FUNCTION_BLOCK "LProcModeSelector"   // FB1708, FBD
TITLE = LModeSelector
{ S7_Optimized_Access := 'FALSE' }
AUTHOR : VCC
FAMILY : Control
NAME : ModeSel
VERSION : 1.0
// ================================================================================
// This module handles that only one mode is selected in the modezon, it also 
// handle interlocking between the HMIs. Each modezone can have 5 HMI.
// ================================================================================
// stored: AutoNumber false, IsIECCheckEnabled false, SetENOAutomatically False, UDAEnableTagReadback false
   VAR_INPUT
      I_StartPB { ExternalAccessible := 'False'; ExternalVisible := 'False'; ExternalWritable := 'False'} : Bool;   // Summary of Start buttons
      I_AlarmResetPB { ExternalAccessible := 'False'; ExternalVisible := 'False'; ExternalWritable := 'False'} : Bool;   // Summary of Alarm reset buttons
      I_SafetyNotOk { ExternalAccessible := 'False'; ExternalVisible := 'False'; ExternalWritable := 'False'} : Bool;   // Safety is not ok
      I_FailSafeResetAck { ExternalAccessible := 'False'; ExternalVisible := 'False'; ExternalWritable := 'False'} : Bool;   // F_Ack_Op FB in safety program is requesting value 9 on FailSafeReset output
      I_FailSafeAckID { ExternalAccessible := 'False'; ExternalVisible := 'False'; ExternalWritable := 'False'} : Int;   // F_Ack ID
      I_HMI1ForceMan { ExternalAccessible := 'False'; ExternalVisible := 'False'; ExternalWritable := 'False'} : Bool;   // Forced manual selected on HMI1
      I_HMI1SetPB { ExternalAccessible := 'False'; ExternalVisible := 'False'; ExternalWritable := 'False'} : Bool;   // Set PB activated on HMI1
      I_HMI1ResetPB { ExternalAccessible := 'False'; ExternalVisible := 'False'; ExternalWritable := 'False'} : Bool;   // Reset PB activated on HMI1
      I_HMI1StartPB { ExternalAccessible := 'False'; ExternalVisible := 'False'; ExternalWritable := 'False'} : Bool;   // Start PB activated on HMI1
      I_HMI1AlarmResetPB { ExternalAccessible := 'False'; ExternalVisible := 'False'; ExternalWritable := 'False'} : Bool;   // AlarmReset PB activated on HMI1
      I_HMI2ForceMan { ExternalAccessible := 'False'; ExternalVisible := 'False'; ExternalWritable := 'False'} : Bool;   // Forced manual selected on HMI2
      I_HMI2SetPB { ExternalAccessible := 'False'; ExternalVisible := 'False'; ExternalWritable := 'False'} : Bool;   // Set PB activated on HMI2
      I_HMI2ResetPB { ExternalAccessible := 'False'; ExternalVisible := 'False'; ExternalWritable := 'False'} : Bool;   // Reset PB activated on HMI2
      I_HMI2StartPB { ExternalAccessible := 'False'; ExternalVisible := 'False'; ExternalWritable := 'False'} : Bool;   // Start PB activated on HMI2
      I_HMI2AlarmResetPB { ExternalAccessible := 'False'; ExternalVisible := 'False'; ExternalWritable := 'False'} : Bool;   // AlarmReset PB activated on HMI2
      I_HMI3ForceMan { ExternalAccessible := 'False'; ExternalVisible := 'False'; ExternalWritable := 'False'} : Bool;   // Forced manual selected on HMI3
      I_HMI3SetPB { ExternalAccessible := 'False'; ExternalVisible := 'False'; ExternalWritable := 'False'} : Bool;   // Set PB activated on HMI3
      I_HMI3ResetPB { ExternalAccessible := 'False'; ExternalVisible := 'False'; ExternalWritable := 'False'} : Bool;   // Reset PB activated on HMI3
      I_HMI3StartPB { ExternalAccessible := 'False'; ExternalVisible := 'False'; ExternalWritable := 'False'} : Bool;   // Start PB activated on HMI
      I_HMI3AlarmResetPB { ExternalAccessible := 'False'; ExternalVisible := 'False'; ExternalWritable := 'False'} : Bool;   // AlarmReset PB activated on HMI3
      I_HMI4ForceMan { ExternalAccessible := 'False'; ExternalVisible := 'False'; ExternalWritable := 'False'} : Bool;   // Forced manual selected on HMI4
      I_HMI4SetPB { ExternalAccessible := 'False'; ExternalVisible := 'False'; ExternalWritable := 'False'} : Bool;   // Set PB activated on HMI4
      I_HMI4ResetPB { ExternalAccessible := 'False'; ExternalVisible := 'False'; ExternalWritable := 'False'} : Bool;   // Reset PB activated on HMI4
      I_HMI4StartPB { ExternalAccessible := 'False'; ExternalVisible := 'False'; ExternalWritable := 'False'} : Bool;   // Start PB activated on HMI4
      I_HMI4AlarmResetPB { ExternalAccessible := 'False'; ExternalVisible := 'False'; ExternalWritable := 'False'} : Bool;   // AlarmReset PB activated on HMI4
      I_HMI5ForceMan { ExternalAccessible := 'False'; ExternalVisible := 'False'; ExternalWritable := 'False'} : Bool;   // Forced manual selected on HMI5
      I_HMI5SetPB { ExternalAccessible := 'False'; ExternalVisible := 'False'; ExternalWritable := 'False'} : Bool;   // Set PB activated on HMI5
      I_HMI5ResetPB { ExternalAccessible := 'False'; ExternalVisible := 'False'; ExternalWritable := 'False'} : Bool;   // Reset PB activated on HMI5
      I_HMI5StartPB { ExternalAccessible := 'False'; ExternalVisible := 'False'; ExternalWritable := 'False'} : Bool;   // Start PB activated on HMI5
      I_HMI5AlarmResetPB { ExternalAccessible := 'False'; ExternalVisible := 'False'; ExternalWritable := 'False'} : Bool;   // AlarmReset PB activated on HMI5
   END_VAR
   VAR_OUTPUT
      O_PBSetPBResetAllAutoSel { ExternalAccessible := 'False'; ExternalVisible := 'False'; ExternalWritable := 'False'} : Struct   // Set PB activated - Reset PB activated - All HMI Auto selected
         HMI1SetPB { ExternalAccessible := 'False'; ExternalVisible := 'False'; ExternalWritable := 'False'} : Bool;   // Set PB activated on HMI1
         HMI1ResetPB { ExternalAccessible := 'False'; ExternalVisible := 'False'; ExternalWritable := 'False'} : Bool;   // Reset PB activated on HMI1
         HMI1AllHMIAutoSel { ExternalAccessible := 'False'; ExternalVisible := 'False'; ExternalWritable := 'False'} : Bool;   // All HMI Auto selected on HMI1
         HMI2SetPB { ExternalAccessible := 'False'; ExternalVisible := 'False'; ExternalWritable := 'False'} : Bool;   // Set PB activated on HMI2
         HMI2ResetPB { ExternalAccessible := 'False'; ExternalVisible := 'False'; ExternalWritable := 'False'} : Bool;   // Reset PB activated on HMI2
         HMI2AllHMIAutoSel { ExternalAccessible := 'False'; ExternalVisible := 'False'; ExternalWritable := 'False'} : Bool;   // All HMI Auto selected on HMI2
         HMI3SetPB { ExternalAccessible := 'False'; ExternalVisible := 'False'; ExternalWritable := 'False'} : Bool;   // Set PB activated on HMI3
         HMI3ResetPB { ExternalAccessible := 'False'; ExternalVisible := 'False'; ExternalWritable := 'False'} : Bool;   // Reset PB activated on HMI3
         HMI3AllHMIAutoSel { ExternalAccessible := 'False'; ExternalVisible := 'False'; ExternalWritable := 'False'} : Bool;   // All HMI Auto selected on HMI3
         HMI4SetPB { ExternalAccessible := 'False'; ExternalVisible := 'False'; ExternalWritable := 'False'} : Bool;   // Set PB activated on HMI4
         HMI4ResetPB { ExternalAccessible := 'False'; ExternalVisible := 'False'; ExternalWritable := 'False'} : Bool;   // Reset PB activated on HMI4
         HMI4AllHMIAutoSel { ExternalAccessible := 'False'; ExternalVisible := 'False'; ExternalWritable := 'False'} : Bool;   // All HMI Auto selected on HMI4
         HMI5SetPB { ExternalAccessible := 'False'; ExternalVisible := 'False'; ExternalWritable := 'False'} : Bool;   // Set PB activated on HMI5
         HMI5ResetPB { ExternalAccessible := 'False'; ExternalVisible := 'False'; ExternalWritable := 'False'} : Bool;   // Reset PB activated on HMI5
         HMI5AllHMIAutoSel { ExternalAccessible := 'False'; ExternalVisible := 'False'; ExternalWritable := 'False'} : Bool;   // All HMI Auto selected on HMI5
         StartPBSel { ExternalAccessible := 'False'; ExternalVisible := 'False'; ExternalWritable := 'False'} : Bool;   // Start is activated
         AlarmResetPBSel { ExternalAccessible := 'False'; ExternalVisible := 'False'; ExternalWritable := 'False'} : Bool;   // Alarm reset is activated
      END_STRUCT;
   END_VAR
   VAR_IN_OUT
      IO_FailsafeReset { ExternalAccessible := 'False'; ExternalVisible := 'False'; ExternalWritable := 'False'} : Int;   // Number to Failsafe to reset safety
   END_VAR
   VAR DB_SPECIFIC
      H_HMIHomeRunModeCmd : Word;   // Homerun Mode commands from HMI
      H_Anim : Word;   // Animation for HMI
      H_ActiveHMI : Int;   // Active HMI
      H_NameActiveHMI : String[25];   // Name of the Active HMI
      H_LockManTime : Int;   // Lock manual time
      H_HMI1ModeCmd : Word;   // Mode commands from HMI1
      H_HMI2ModeCmd : Word;   // Mode commands from HMI2
      H_HMI3ModeCmd : Word;   // Mode commands from HMI3
      H_HMI4ModeCmd : Word;   // Mode commands from HMI4
      H_HMI5ModeCmd : Word;   // Mode commands from HMI5. For operator panels, no S7_m_c
      HMI1AutoSel { ExternalAccessible := 'False'; ExternalVisible := 'False'; ExternalWritable := 'False'} : Bool;   // Auto selected on HMI1
      HMI1StepSel { ExternalAccessible := 'False'; ExternalVisible := 'False'; ExternalWritable := 'False'} : Bool;   // Step selected on HMI1
      HMI1HomeRunSel { ExternalAccessible := 'False'; ExternalVisible := 'False'; ExternalWritable := 'False'} : Bool;   // Homerun selected on HMI1
      HMI1ManualSel { ExternalAccessible := 'False'; ExternalVisible := 'False'; ExternalWritable := 'False'} : Bool;   // Manual selected on HMI1
      HMI1LockManual { ExternalAccessible := 'False'; ExternalVisible := 'False'; ExternalWritable := 'False'} : Bool;   // Lock manual for HMI1
      HMI1AllHMIAutoSel { ExternalAccessible := 'False'; ExternalVisible := 'False'; ExternalWritable := 'False'} : Bool;   // All HMI Auto selected on HMI1
      HMI1Start { ExternalAccessible := 'False'; ExternalVisible := 'False'; ExternalWritable := 'False'} : Bool;   // Start on HMI1
      HMI1AlarmReset { ExternalAccessible := 'False'; ExternalVisible := 'False'; ExternalWritable := 'False'} : Bool;   // AlarmReset on HMI1
      HMI1ResetTM { ExternalAccessible := 'False'; ExternalVisible := 'False'; ExternalWritable := 'False'} : Bool;   // Reset transport memory from HMI1
      HMI1ResetSeq { ExternalAccessible := 'False'; ExternalVisible := 'False'; ExternalWritable := 'False'} : Bool;   // Reset sequence from HMI1
      HMI1CycleFinished { ExternalAccessible := 'False'; ExternalVisible := 'False'; ExternalWritable := 'False'} : Bool;   // Cycle Finished from HMI1
      HMI1AlarmResetAck { ExternalAccessible := 'False'; ExternalVisible := 'False'; ExternalWritable := 'False'} : Bool;   // Alarm Reset acknowledge from HMI1
      HMI2AutoSel { ExternalAccessible := 'False'; ExternalVisible := 'False'; ExternalWritable := 'False'} : Bool;   // Auto selected on HMI2
      HMI2StepSel { ExternalAccessible := 'False'; ExternalVisible := 'False'; ExternalWritable := 'False'} : Bool;   // Step selected on HMI2
      HMI2HomeRunSel { ExternalAccessible := 'False'; ExternalVisible := 'False'; ExternalWritable := 'False'} : Bool;   // Homerun selected on HMI2
      HMI2ManualSel { ExternalAccessible := 'False'; ExternalVisible := 'False'; ExternalWritable := 'False'} : Bool;   // Manual selected on HMI2
      HMI2LockManual { ExternalAccessible := 'False'; ExternalVisible := 'False'; ExternalWritable := 'False'} : Bool;   // Lock manual for HMI2
      HMI2AllHMIAutoSel { ExternalAccessible := 'False'; ExternalVisible := 'False'; ExternalWritable := 'False'} : Bool;   // All HMI Auto selected on HMI2
      HMI2Start { ExternalAccessible := 'False'; ExternalVisible := 'False'; ExternalWritable := 'False'} : Bool;   // Start on HMI2
      HMI2AlarmReset { ExternalAccessible := 'False'; ExternalVisible := 'False'; ExternalWritable := 'False'} : Bool;   // AlarmReset on HMI2
      HMI2ResetTM { ExternalAccessible := 'False'; ExternalVisible := 'False'; ExternalWritable := 'False'} : Bool;   // Reset transport memory from HMI2
      HMI2ResetSeq { ExternalAccessible := 'False'; ExternalVisible := 'False'; ExternalWritable := 'False'} : Bool;   // Reset sequence from HMI2
      HMI2CycleFinished { ExternalAccessible := 'False'; ExternalVisible := 'False'; ExternalWritable := 'False'} : Bool;   // Cycle Finished from HMI2
      HMI2AlarmResetAck { ExternalAccessible := 'False'; ExternalVisible := 'False'; ExternalWritable := 'False'} : Bool;   // Alarm Reset acknowledge from HMI2
      HMI3AutoSel { ExternalAccessible := 'False'; ExternalVisible := 'False'; ExternalWritable := 'False'} : Bool;   // Auto selected on HMI3
      HMI3StepSel { ExternalAccessible := 'False'; ExternalVisible := 'False'; ExternalWritable := 'False'} : Bool;   // Step selected on HMI3
      HMI3HomeRunSel { ExternalAccessible := 'False'; ExternalVisible := 'False'; ExternalWritable := 'False'} : Bool;   // Homerun selected on HMI3
      HMI3ManualSel { ExternalAccessible := 'False'; ExternalVisible := 'False'; ExternalWritable := 'False'} : Bool;   // Manual selected on HMI3
      HMI3LockManual { ExternalAccessible := 'False'; ExternalVisible := 'False'; ExternalWritable := 'False'} : Bool;   // Lock manual for HMI3
      HMI3AllHMIAutoSel { ExternalAccessible := 'False'; ExternalVisible := 'False'; ExternalWritable := 'False'} : Bool;   // All HMI Auto selected on HMI3
      HMI3Start { ExternalAccessible := 'False'; ExternalVisible := 'False'; ExternalWritable := 'False'} : Bool;   // Start on HMI3
      HMI3AlarmReset { ExternalAccessible := 'False'; ExternalVisible := 'False'; ExternalWritable := 'False'} : Bool;   // AlarmReset on HMI3
      HMI3ResetTM { ExternalAccessible := 'False'; ExternalVisible := 'False'; ExternalWritable := 'False'} : Bool;   // Reset transport memory from HMI3
      HMI3ResetSeq { ExternalAccessible := 'False'; ExternalVisible := 'False'; ExternalWritable := 'False'} : Bool;   // Reset sequence from HMI3
      HMI3CycleFinished { ExternalAccessible := 'False'; ExternalVisible := 'False'; ExternalWritable := 'False'} : Bool;   // Cycle Finished from HMI3
      HMI3AlarmResetAck { ExternalAccessible := 'False'; ExternalVisible := 'False'; ExternalWritable := 'False'} : Bool;   // Alarm Reset acknowledge from 3
      HMI4AutoSel { ExternalAccessible := 'False'; ExternalVisible := 'False'; ExternalWritable := 'False'} : Bool;   // Auto selected on HMI4
      HMI4StepSel { ExternalAccessible := 'False'; ExternalVisible := 'False'; ExternalWritable := 'False'} : Bool;   // Step selected on HMI4
      HMI4HomeRunSel { ExternalAccessible := 'False'; ExternalVisible := 'False'; ExternalWritable := 'False'} : Bool;   // Homerun selected on HMI4
      HMI4ManualSel { ExternalAccessible := 'False'; ExternalVisible := 'False'; ExternalWritable := 'False'} : Bool;   // Manual selected on HMI4
      HMI4LockManual { ExternalAccessible := 'False'; ExternalVisible := 'False'; ExternalWritable := 'False'} : Bool;   // Lock manual for HMI4
      HMI4AllHMIAutoSel { ExternalAccessible := 'False'; ExternalVisible := 'False'; ExternalWritable := 'False'} : Bool;   // All HMI Auto selected on HMI4
      HMI4Start { ExternalAccessible := 'False'; ExternalVisible := 'False'; ExternalWritable := 'False'} : Bool;   // Start on HMI4
      HMI4AlarmReset { ExternalAccessible := 'False'; ExternalVisible := 'False'; ExternalWritable := 'False'} : Bool;   // AlarmReset on HMI4
      HMI4ResetTM { ExternalAccessible := 'False'; ExternalVisible := 'False'; ExternalWritable := 'False'} : Bool;   // Reset transport memory from HMI4
      HMI4ResetSeq { ExternalAccessible := 'False'; ExternalVisible := 'False'; ExternalWritable := 'False'} : Bool;   // Reset sequence from HMI4
      HMI4CycleFinished { ExternalAccessible := 'False'; ExternalVisible := 'False'; ExternalWritable := 'False'} : Bool;   // Cycle Finished from HMI4
      HMI4AlarmResetAck { ExternalAccessible := 'False'; ExternalVisible := 'False'; ExternalWritable := 'False'} : Bool;   // Alarm Reset acknowledge from HMI4
      HMI5AutoSel { ExternalAccessible := 'False'; ExternalVisible := 'False'; ExternalWritable := 'False'} : Bool;   // Auto selected on HMI5
      HMI5StepSel { ExternalAccessible := 'False'; ExternalVisible := 'False'; ExternalWritable := 'False'} : Bool;   // Step selected on HMI5
      HMI5HomeRunSel { ExternalAccessible := 'False'; ExternalVisible := 'False'; ExternalWritable := 'False'} : Bool;   // Homerun selected on HMI5
      HMI5ManualSel { ExternalAccessible := 'False'; ExternalVisible := 'False'; ExternalWritable := 'False'} : Bool;   // Manual selected on HMI5
      HMI5LockManual { ExternalAccessible := 'False'; ExternalVisible := 'False'; ExternalWritable := 'False'} : Bool;   // Lock manual for HMI5
      HMI5AllHMIAutoSel { ExternalAccessible := 'False'; ExternalVisible := 'False'; ExternalWritable := 'False'} : Bool;   // All HMI Auto selected on HMI5
      HMI5Start { ExternalAccessible := 'False'; ExternalVisible := 'False'; ExternalWritable := 'False'} : Bool;   // Start on HMI5
      HMI5AlarmReset { ExternalAccessible := 'False'; ExternalVisible := 'False'; ExternalWritable := 'False'} : Bool;   // AlarmReset on HMI5
      HMI5ResetTM { ExternalAccessible := 'False'; ExternalVisible := 'False'; ExternalWritable := 'False'} : Bool;   // Reset transport memory from HMI5
      HMI5ResetSeq { ExternalAccessible := 'False'; ExternalVisible := 'False'; ExternalWritable := 'False'} : Bool;   // Reset sequence from HMI5
      HMI5CycleFinished { ExternalAccessible := 'False'; ExternalVisible := 'False'; ExternalWritable := 'False'} : Bool;   // Cycle Finished from HMI5
      HMI5AlarmResetAck { ExternalAccessible := 'False'; ExternalVisible := 'False'; ExternalWritable := 'False'} : Bool;   // Alarm Reset acknowledge from HMI5
      HMIHomeRunRedo { ExternalAccessible := 'False'; ExternalVisible := 'False'; ExternalWritable := 'False'} : Bool;   // Redo after homerun from HMI
      HMIHomeRunWorkDone { ExternalAccessible := 'False'; ExternalVisible := 'False'; ExternalWritable := 'False'} : Bool;   // WorkDone after homerun from HMI
      LockManualTimeout { ExternalAccessible := 'False'; ExternalVisible := 'False'; ExternalWritable := 'False'} : Bool;   // Lock manual button timeout
      AllHmiAutoSel { ExternalAccessible := 'False'; ExternalVisible := 'False'; ExternalWritable := 'False'} : Bool;   // All Hmi Auto selected
      AlarmResetPBSel { ExternalAccessible := 'False'; ExternalVisible := 'False'; ExternalWritable := 'False'} : Bool;   // Alarm reset is activated
      AlarmResetPBSelReset { ExternalAccessible := 'False'; ExternalVisible := 'False'; ExternalWritable := 'False'} : Bool;   // Reset AlarmResetPBSel after predefined time
      AlarmResetPBSelResetPE { ExternalAccessible := 'False'; ExternalVisible := 'False'; ExternalWritable := 'False'} : Bool;   // Positive edge of AlarmResetPbSelReset
      FailSafeReset6Pulse { ExternalAccessible := 'False'; ExternalVisible := 'False'; ExternalWritable := 'False'} : Bool;   // Pulse to set value 6 on FailSafeReset Output
      FailSafeReset9Pulse { ExternalAccessible := 'False'; ExternalVisible := 'False'; ExternalWritable := 'False'} : Bool;   // Pulse to set value 9 on FailSafeReset Output
      ResetAlarmAckMemPulse { ExternalAccessible := 'False'; ExternalVisible := 'False'; ExternalWritable := 'False'} : Bool;   // Pulse to reset AlarmResetAckMem on negative edge of I_FailSafeResetAck
      AlarmResetAckMem { ExternalAccessible := 'False'; ExternalVisible := 'False'; ExternalWritable := 'False'} : Bool;   // memory : Pushbutton AlarmResetAck has been pushed on HMI
      StartPBSel { ExternalAccessible := 'False'; ExternalVisible := 'False'; ExternalWritable := 'False'} : Bool;   // Summary of the Start push buttons
      HMIStartPE { ExternalAccessible := 'False'; ExternalVisible := 'False'; ExternalWritable := 'False'} : Bool;   // Positive edge on start button from HMI
      HMIResetTMPE { ExternalAccessible := 'False'; ExternalVisible := 'False'; ExternalWritable := 'False'} : Bool;   // Positive edge on ResetTM button from HMI
      HMIResetSeqPE { ExternalAccessible := 'False'; ExternalVisible := 'False'; ExternalWritable := 'False'} : Bool;   // Positive edge on ResetSeq button from HMI
      HMIAlarmResetAckPE { ExternalAccessible := 'False'; ExternalVisible := 'False'; ExternalWritable := 'False'} : Bool;   // Positive edge on AlarmResetAck button from HMI
      HMILockManualPE { ExternalAccessible := 'False'; ExternalVisible := 'False'; ExternalWritable := 'False'} : Bool;   // Positive edge on LockManual button from HMI
      FailsafeReset { ExternalAccessible := 'False'; ExternalVisible := 'False'; ExternalWritable := 'False'} : Int;   // Number to Failsafe to reset safety
      ActiveHMI { ExternalAccessible := 'False'; ExternalVisible := 'False'; ExternalWritable := 'False'} : Int;   // Help memory for Active HMI
   END_VAR
   VAR
      TimerLockMan { ExternalAccessible := 'False'; ExternalVisible := 'False'; ExternalWritable := 'False'; S7_SetPoint := 'True'} : "LTimer";   // Timer on Lock manual
      TimerAlarmResetPB { ExternalAccessible := 'False'; ExternalVisible := 'False'; ExternalWritable := 'False'; S7_SetPoint := 'True'} : "LTimer";   // Timer on alarm reset
   END_VAR
   VAR_TEMP
      PHMI1AutoSel : Bool;   // Pulse Auto selected HMI1
      PHMI2AutoSel : Bool;   // Pulse Auto selected HMI2
      PHMI3AutoSel : Bool;   // Pulse Auto selected HMI3
      PHMI4AutoSel : Bool;   // Pulse Auto selected HMI4
      PHMI5AutoSel : Bool;   // Pulse Auto selected HMI5
   END_VAR
   VAR_TEMP   // added for the SCL form of the ladder/FBD networks
      _w1 : Bool;
      _w2 : Bool;
      _w3 : Bool;
      _w4 : Bool;
      _w5 : Bool;
   END_VAR
BEGIN

REGION Network 1: **** 1 - Inputs **** Extract the modeselection from HMI 1
   // Extract the modeselection from HMI 1
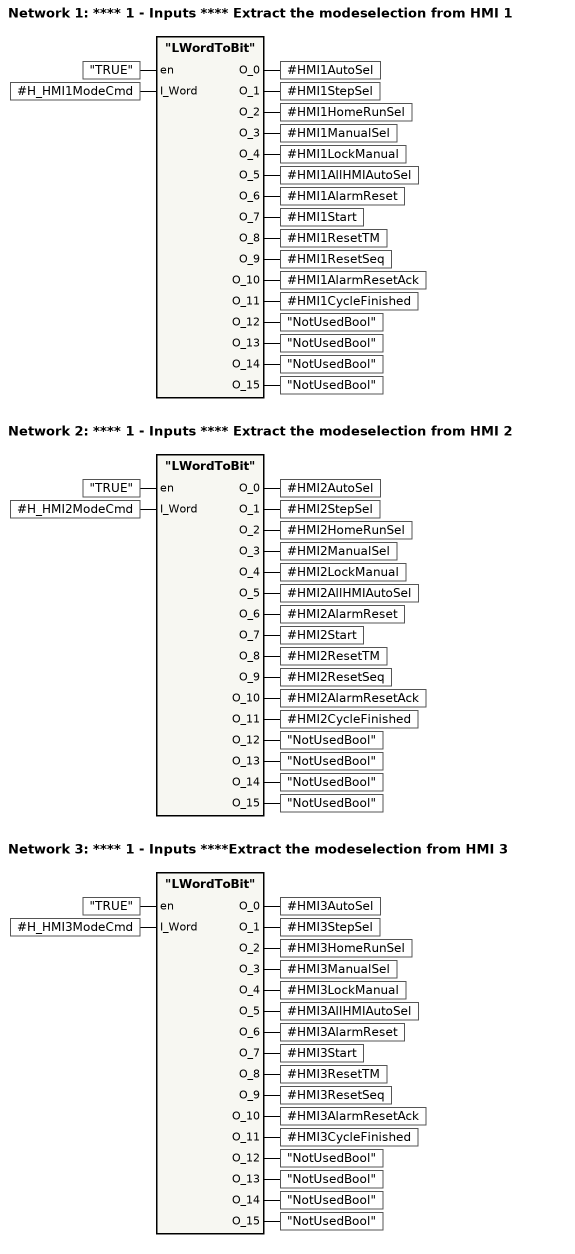
   IF "TRUE" THEN
       "LWordToBit"(I_Word := #H_HMI1ModeCmd,
                    O_0 => #HMI1AutoSel,
                    O_1 => #HMI1StepSel,
                    O_2 => #HMI1HomeRunSel,
                    O_3 => #HMI1ManualSel,
                    O_4 => #HMI1LockManual,
                    O_5 => #HMI1AllHMIAutoSel,
                    O_6 => #HMI1AlarmReset,
                    O_7 => #HMI1Start,
                    O_8 => #HMI1ResetTM,
                    O_9 => #HMI1ResetSeq,
                    O_10 => #HMI1AlarmResetAck,
                    O_11 => #HMI1CycleFinished,
                    O_12 => "NotUsedBool",
                    O_13 => "NotUsedBool",
                    O_14 => "NotUsedBool",
                    O_15 => "NotUsedBool");
   END_IF;
END_REGION

REGION Network 2: **** 1 - Inputs **** Extract the modeselection from HMI 2
   // Extract the modeselection from HMI 2
   IF "TRUE" THEN
       "LWordToBit"(I_Word := #H_HMI2ModeCmd,
                    O_0 => #HMI2AutoSel,
                    O_1 => #HMI2StepSel,
                    O_2 => #HMI2HomeRunSel,
                    O_3 => #HMI2ManualSel,
                    O_4 => #HMI2LockManual,
                    O_5 => #HMI2AllHMIAutoSel,
                    O_6 => #HMI2AlarmReset,
                    O_7 => #HMI2Start,
                    O_8 => #HMI2ResetTM,
                    O_9 => #HMI2ResetSeq,
                    O_10 => #HMI2AlarmResetAck,
                    O_11 => #HMI2CycleFinished,
                    O_12 => "NotUsedBool",
                    O_13 => "NotUsedBool",
                    O_14 => "NotUsedBool",
                    O_15 => "NotUsedBool");
   END_IF;
END_REGION

REGION Network 3: **** 1 - Inputs ****Extract the modeselection from HMI 3
   // Extract the modeselection from HMI 3
   IF "TRUE" THEN
       "LWordToBit"(I_Word := #H_HMI3ModeCmd,
                    O_0 => #HMI3AutoSel,
                    O_1 => #HMI3StepSel,
                    O_2 => #HMI3HomeRunSel,
                    O_3 => #HMI3ManualSel,
                    O_4 => #HMI3LockManual,
                    O_5 => #HMI3AllHMIAutoSel,
                    O_6 => #HMI3AlarmReset,
                    O_7 => #HMI3Start,
                    O_8 => #HMI3ResetTM,
                    O_9 => #HMI3ResetSeq,
                    O_10 => #HMI3AlarmResetAck,
                    O_11 => #HMI3CycleFinished,
                    O_12 => "NotUsedBool",
                    O_13 => "NotUsedBool",
                    O_14 => "NotUsedBool",
                    O_15 => "NotUsedBool");
   END_IF;
END_REGION

REGION Network 4: **** 1 - Inputs **** Extract the modeselection from HMI 4
   // Extract the modeselection from HMI 4
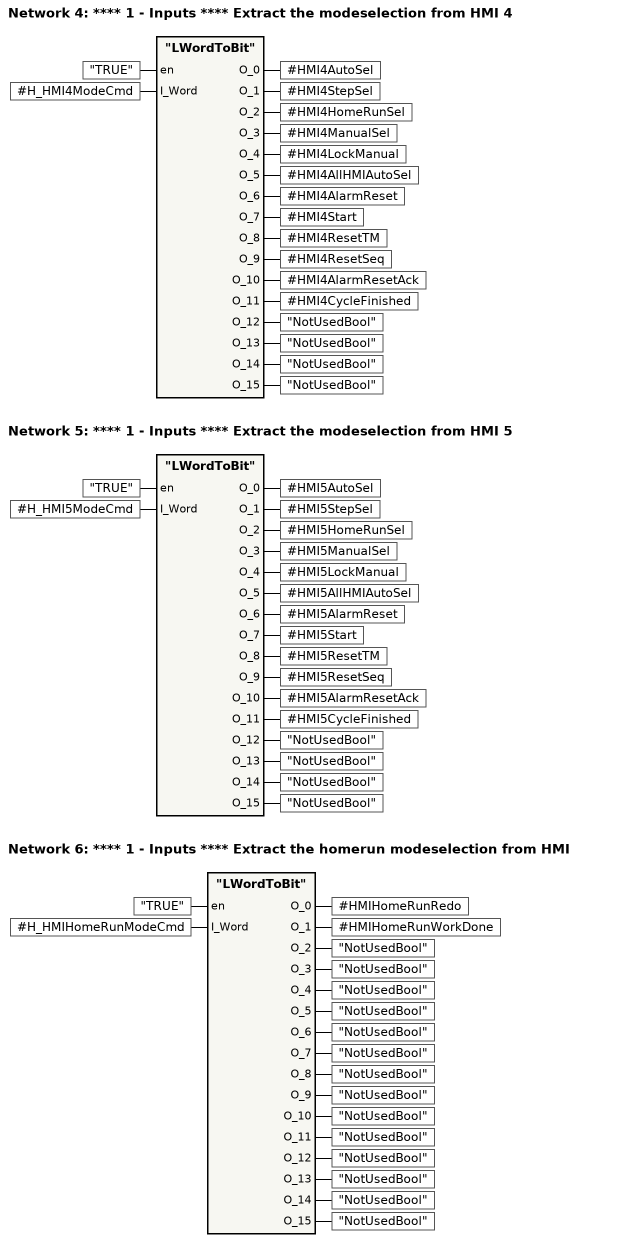
   IF "TRUE" THEN
       "LWordToBit"(I_Word := #H_HMI4ModeCmd,
                    O_0 => #HMI4AutoSel,
                    O_1 => #HMI4StepSel,
                    O_2 => #HMI4HomeRunSel,
                    O_3 => #HMI4ManualSel,
                    O_4 => #HMI4LockManual,
                    O_5 => #HMI4AllHMIAutoSel,
                    O_6 => #HMI4AlarmReset,
                    O_7 => #HMI4Start,
                    O_8 => #HMI4ResetTM,
                    O_9 => #HMI4ResetSeq,
                    O_10 => #HMI4AlarmResetAck,
                    O_11 => #HMI4CycleFinished,
                    O_12 => "NotUsedBool",
                    O_13 => "NotUsedBool",
                    O_14 => "NotUsedBool",
                    O_15 => "NotUsedBool");
   END_IF;
END_REGION

REGION Network 5: **** 1 - Inputs **** Extract the modeselection from HMI 5
   // Extract the modeselection from HMI 5
   IF "TRUE" THEN
       "LWordToBit"(I_Word := #H_HMI5ModeCmd,
                    O_0 => #HMI5AutoSel,
                    O_1 => #HMI5StepSel,
                    O_2 => #HMI5HomeRunSel,
                    O_3 => #HMI5ManualSel,
                    O_4 => #HMI5LockManual,
                    O_5 => #HMI5AllHMIAutoSel,
                    O_6 => #HMI5AlarmReset,
                    O_7 => #HMI5Start,
                    O_8 => #HMI5ResetTM,
                    O_9 => #HMI5ResetSeq,
                    O_10 => #HMI5AlarmResetAck,
                    O_11 => #HMI5CycleFinished,
                    O_12 => "NotUsedBool",
                    O_13 => "NotUsedBool",
                    O_14 => "NotUsedBool",
                    O_15 => "NotUsedBool");
   END_IF;
END_REGION

REGION Network 6: **** 1 - Inputs **** Extract the homerun modeselection from HMI
   // Extract the homerun modeselection from HMI
   IF "TRUE" THEN
       "LWordToBit"(I_Word := #H_HMIHomeRunModeCmd,
                    O_0 => #HMIHomeRunRedo,
                    O_1 => #HMIHomeRunWorkDone,
                    O_2 => "NotUsedBool",
                    O_3 => "NotUsedBool",
                    O_4 => "NotUsedBool",
                    O_5 => "NotUsedBool",
                    O_6 => "NotUsedBool",
                    O_7 => "NotUsedBool",
                    O_8 => "NotUsedBool",
                    O_9 => "NotUsedBool",
                    O_10 => "NotUsedBool",
                    O_11 => "NotUsedBool",
                    O_12 => "NotUsedBool",
                    O_13 => "NotUsedBool",
                    O_14 => "NotUsedBool",
                    O_15 => "NotUsedBool");
   END_IF;
END_REGION

REGION Network 7: **** 1 - Inputs **** All HMI Auto selected
   // All HMI Auto selected
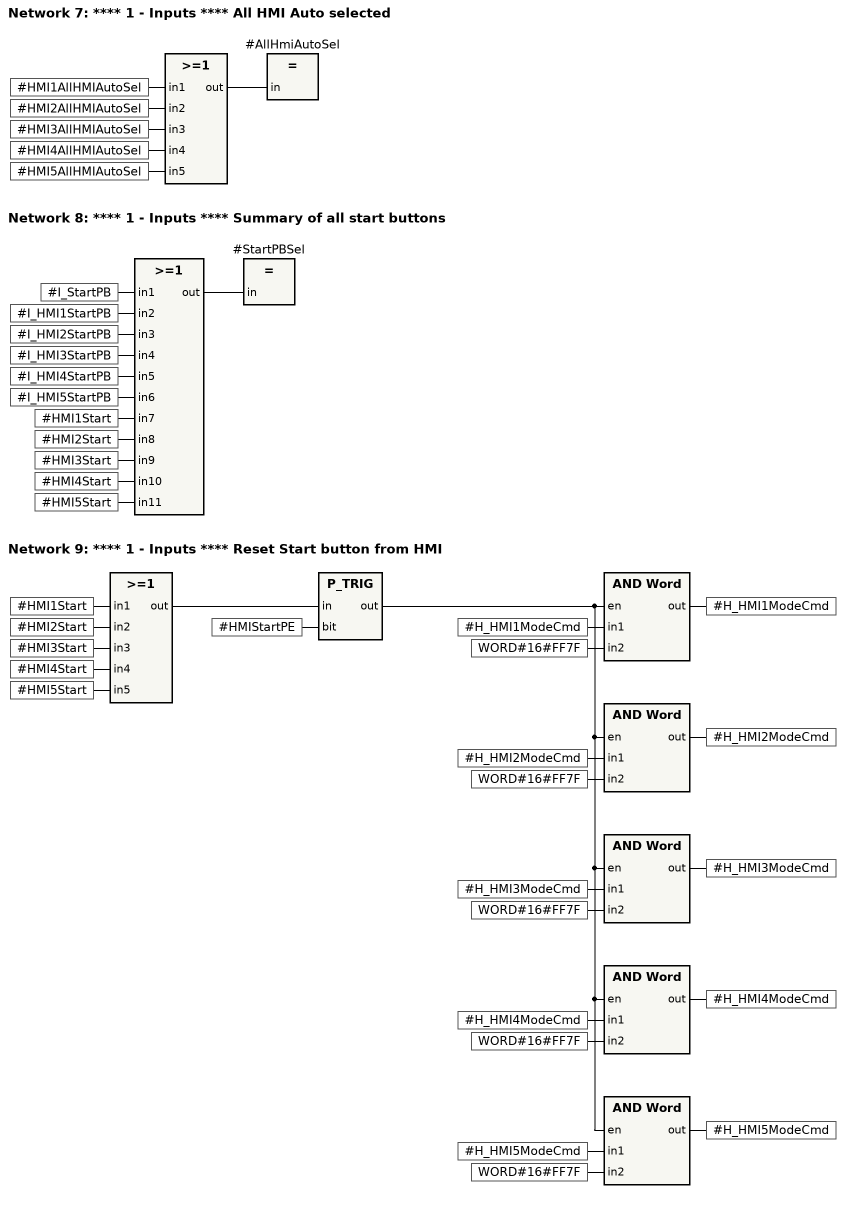
   #AllHmiAutoSel := #HMI1AllHMIAutoSel OR #HMI2AllHMIAutoSel OR #HMI3AllHMIAutoSel OR #HMI4AllHMIAutoSel OR #HMI5AllHMIAutoSel;
END_REGION

REGION Network 8: **** 1 - Inputs **** Summary of all start buttons
   // Summary of all start buttons
   #StartPBSel := #I_StartPB OR #I_HMI1StartPB OR #I_HMI2StartPB OR #I_HMI3StartPB OR #I_HMI4StartPB OR #I_HMI5StartPB OR #HMI1Start OR #HMI2Start OR #HMI3Start OR #HMI4Start OR #HMI5Start;
END_REGION

REGION Network 9: **** 1 - Inputs **** Reset Start button from HMI
   // Reset Start button from HMI
   #_w1 := #HMI1Start OR #HMI2Start OR #HMI3Start OR #HMI4Start OR #HMI5Start;
   #_w2 := #_w1 AND NOT #HMIStartPE;   // rising edge
   #HMIStartPE := #_w1;
   IF #_w2 THEN
       #H_HMI1ModeCmd := #H_HMI1ModeCmd AND WORD#16#FF7F;
       #H_HMI2ModeCmd := #H_HMI2ModeCmd AND WORD#16#FF7F;
       #H_HMI3ModeCmd := #H_HMI3ModeCmd AND WORD#16#FF7F;
       #H_HMI4ModeCmd := #H_HMI4ModeCmd AND WORD#16#FF7F;
       #H_HMI5ModeCmd := #H_HMI5ModeCmd AND WORD#16#FF7F;
   END_IF;
END_REGION

REGION Network 10: **** 1 - Inputs **** Summary of all alarm reset buttons
   // Summary of all alarm reset buttons
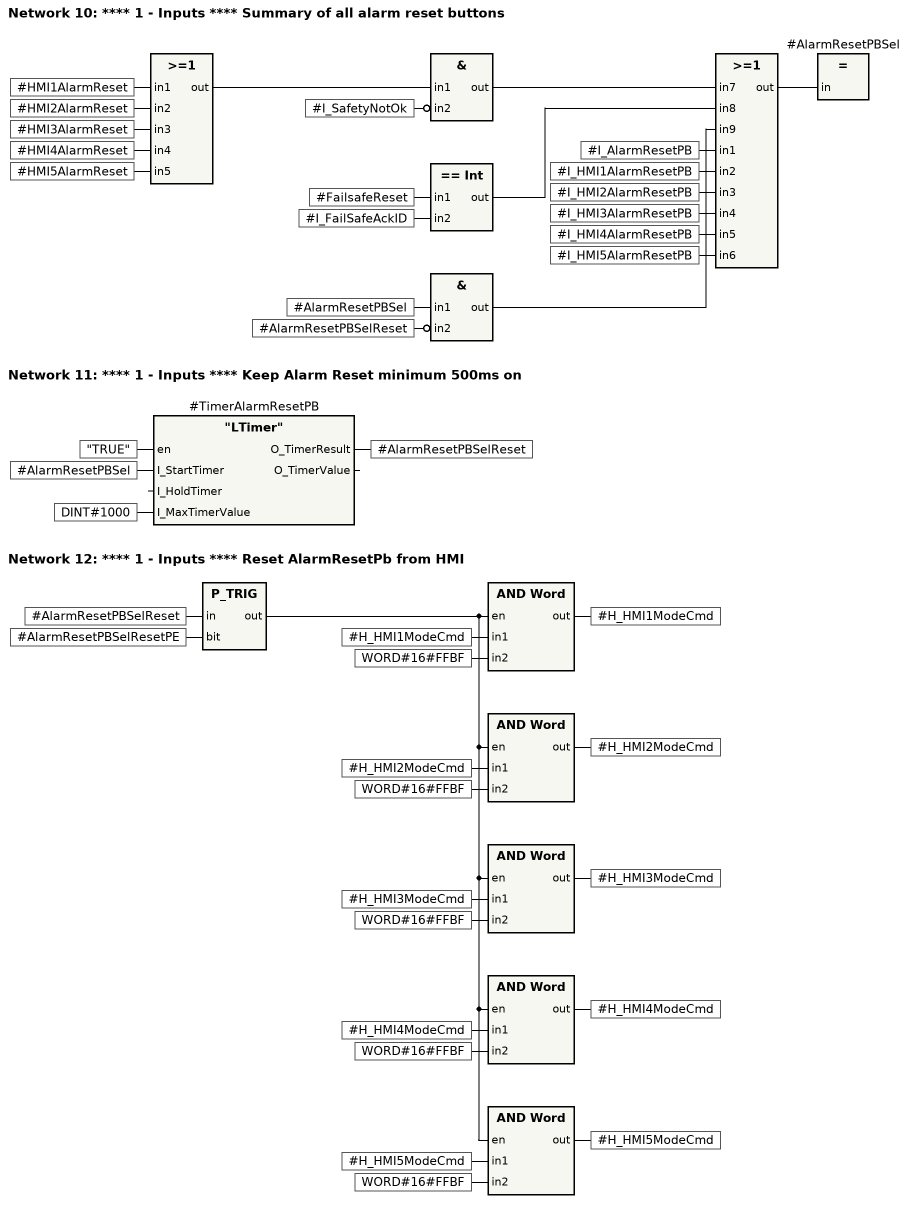
   #AlarmResetPBSel := ((#HMI1AlarmReset OR #HMI2AlarmReset OR #HMI3AlarmReset OR #HMI4AlarmReset OR #HMI5AlarmReset) AND NOT #I_SafetyNotOk) OR (#FailsafeReset = #I_FailSafeAckID) OR (#AlarmResetPBSel AND NOT #AlarmResetPBSelReset) OR #I_AlarmResetPB OR #I_HMI1AlarmResetPB OR #I_HMI2AlarmResetPB OR #I_HMI3AlarmResetPB OR #I_HMI4AlarmResetPB OR #I_HMI5AlarmResetPB;
END_REGION

REGION Network 11: **** 1 - Inputs **** Keep Alarm Reset minimum 500ms on
   // Keep Alarm Reset minimum 500ms on
   IF "TRUE" THEN
       #TimerAlarmResetPB(I_StartTimer := #AlarmResetPBSel,   // "LTimer"
                          I_MaxTimerValue := DINT#1000,
                          O_TimerResult => #AlarmResetPBSelReset);
   END_IF;
END_REGION

REGION Network 12: **** 1 - Inputs **** Reset AlarmResetPb from HMI
   // Reset AlarmResetPb from HMI
   #_w1 := #AlarmResetPBSelReset AND NOT #AlarmResetPBSelResetPE;   // rising edge
   #AlarmResetPBSelResetPE := #AlarmResetPBSelReset;
   IF #_w1 THEN
       #H_HMI1ModeCmd := #H_HMI1ModeCmd AND WORD#16#FFBF;
       #H_HMI2ModeCmd := #H_HMI2ModeCmd AND WORD#16#FFBF;
       #H_HMI3ModeCmd := #H_HMI3ModeCmd AND WORD#16#FFBF;
       #H_HMI4ModeCmd := #H_HMI4ModeCmd AND WORD#16#FFBF;
       #H_HMI5ModeCmd := #H_HMI5ModeCmd AND WORD#16#FFBF;
   END_IF;
END_REGION

REGION Network 13: **** 1 - Inputs **** Reset AlarmResetAckPb from HMI
   // Reset AlarmResetAckPb from HMI
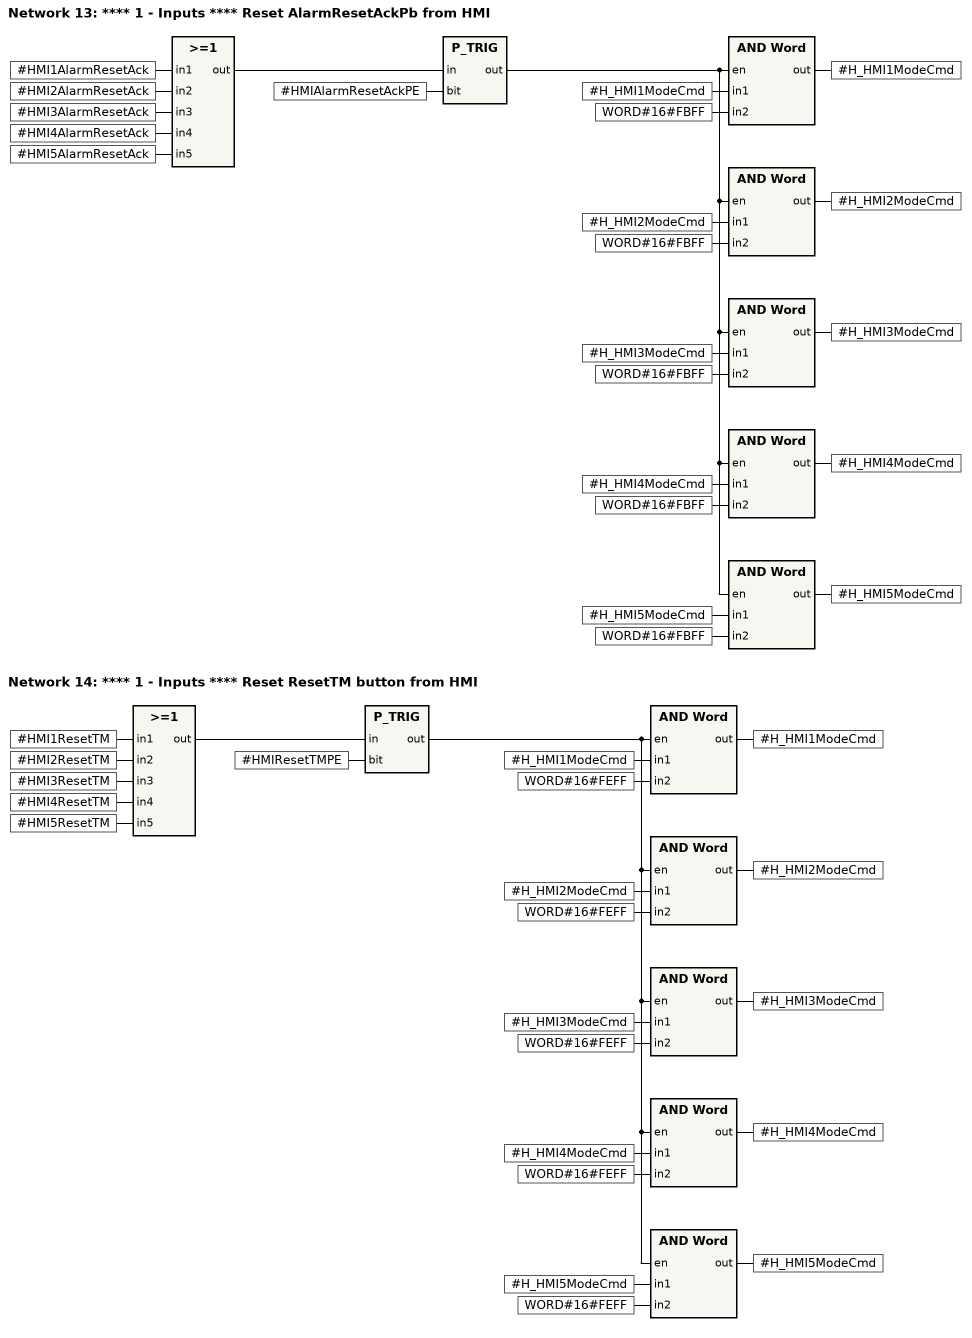
   #_w1 := #HMI1AlarmResetAck OR #HMI2AlarmResetAck OR #HMI3AlarmResetAck OR #HMI4AlarmResetAck OR #HMI5AlarmResetAck;
   #_w2 := #_w1 AND NOT #HMIAlarmResetAckPE;   // rising edge
   #HMIAlarmResetAckPE := #_w1;
   IF #_w2 THEN
       #H_HMI1ModeCmd := #H_HMI1ModeCmd AND WORD#16#FBFF;
       #H_HMI2ModeCmd := #H_HMI2ModeCmd AND WORD#16#FBFF;
       #H_HMI3ModeCmd := #H_HMI3ModeCmd AND WORD#16#FBFF;
       #H_HMI4ModeCmd := #H_HMI4ModeCmd AND WORD#16#FBFF;
       #H_HMI5ModeCmd := #H_HMI5ModeCmd AND WORD#16#FBFF;
   END_IF;
END_REGION

REGION Network 14: **** 1 - Inputs **** Reset ResetTM button from HMI
   // Reset ResetTM button from HMI
   #_w1 := #HMI1ResetTM OR #HMI2ResetTM OR #HMI3ResetTM OR #HMI4ResetTM OR #HMI5ResetTM;
   #_w2 := #_w1 AND NOT #HMIResetTMPE;   // rising edge
   #HMIResetTMPE := #_w1;
   IF #_w2 THEN
       #H_HMI1ModeCmd := #H_HMI1ModeCmd AND WORD#16#FEFF;
       #H_HMI2ModeCmd := #H_HMI2ModeCmd AND WORD#16#FEFF;
       #H_HMI3ModeCmd := #H_HMI3ModeCmd AND WORD#16#FEFF;
       #H_HMI4ModeCmd := #H_HMI4ModeCmd AND WORD#16#FEFF;
       #H_HMI5ModeCmd := #H_HMI5ModeCmd AND WORD#16#FEFF;
   END_IF;
END_REGION

REGION Network 15: **** 1 - Inputs **** Reset ResetSeq button from HMI
   // Reset ResetSeq button from HMI
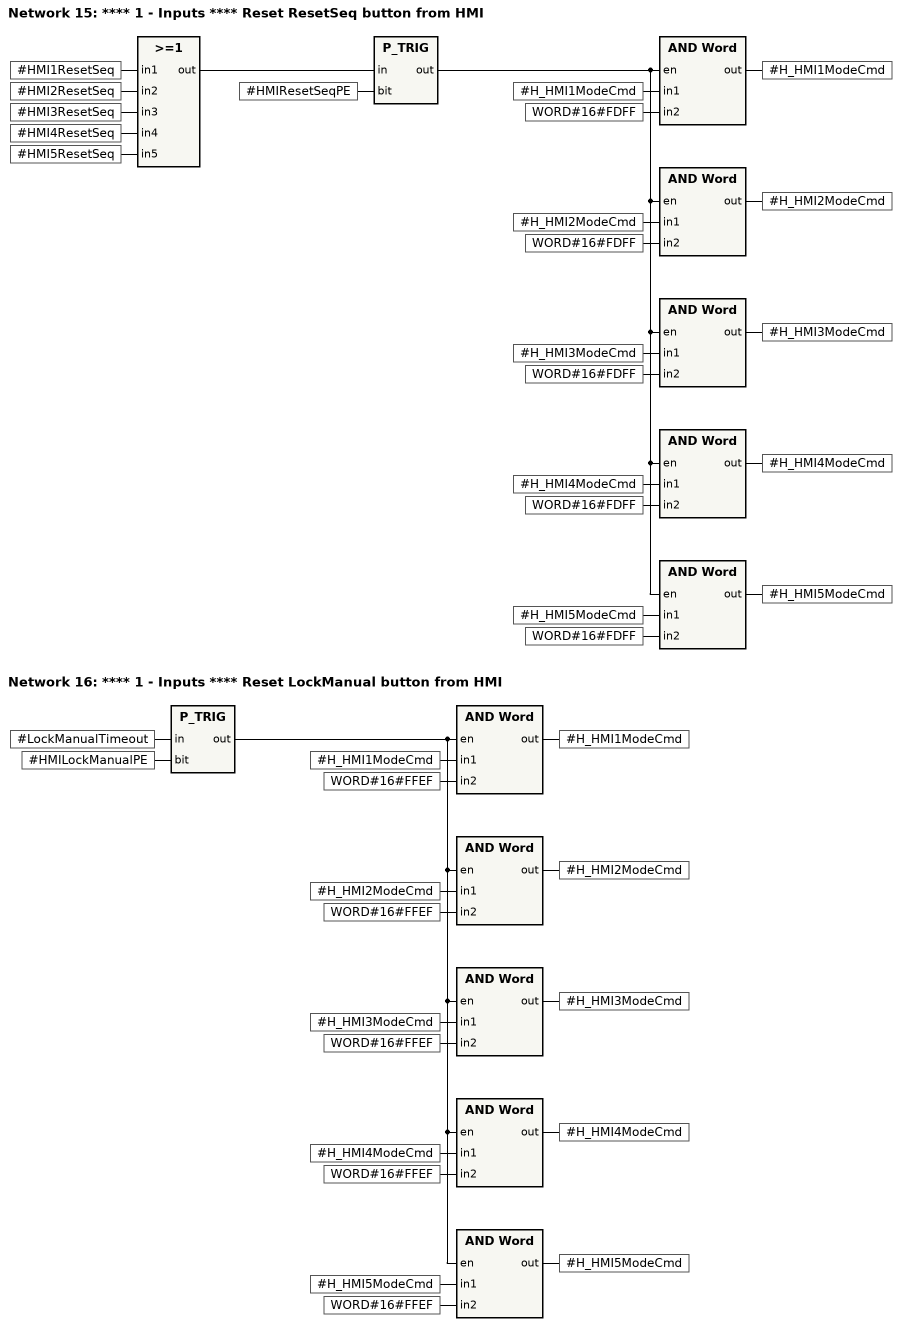
   #_w1 := #HMI1ResetSeq OR #HMI2ResetSeq OR #HMI3ResetSeq OR #HMI4ResetSeq OR #HMI5ResetSeq;
   #_w2 := #_w1 AND NOT #HMIResetSeqPE;   // rising edge
   #HMIResetSeqPE := #_w1;
   IF #_w2 THEN
       #H_HMI1ModeCmd := #H_HMI1ModeCmd AND WORD#16#FDFF;
       #H_HMI2ModeCmd := #H_HMI2ModeCmd AND WORD#16#FDFF;
       #H_HMI3ModeCmd := #H_HMI3ModeCmd AND WORD#16#FDFF;
       #H_HMI4ModeCmd := #H_HMI4ModeCmd AND WORD#16#FDFF;
       #H_HMI5ModeCmd := #H_HMI5ModeCmd AND WORD#16#FDFF;
   END_IF;
END_REGION

REGION Network 16: **** 1 - Inputs **** Reset LockManual button from HMI
   // Reset LockManual button from HMI
   #_w1 := #LockManualTimeout AND NOT #HMILockManualPE;   // rising edge
   #HMILockManualPE := #LockManualTimeout;
   IF #_w1 THEN
       #H_HMI1ModeCmd := #H_HMI1ModeCmd AND WORD#16#FFEF;
       #H_HMI2ModeCmd := #H_HMI2ModeCmd AND WORD#16#FFEF;
       #H_HMI3ModeCmd := #H_HMI3ModeCmd AND WORD#16#FFEF;
       #H_HMI4ModeCmd := #H_HMI4ModeCmd AND WORD#16#FFEF;
       #H_HMI5ModeCmd := #H_HMI5ModeCmd AND WORD#16#FFEF;
   END_IF;
END_REGION

REGION Network 17: **** 4.5 - Machine Status - Modes **** Reset activ HMI
   // Reset activ HMI
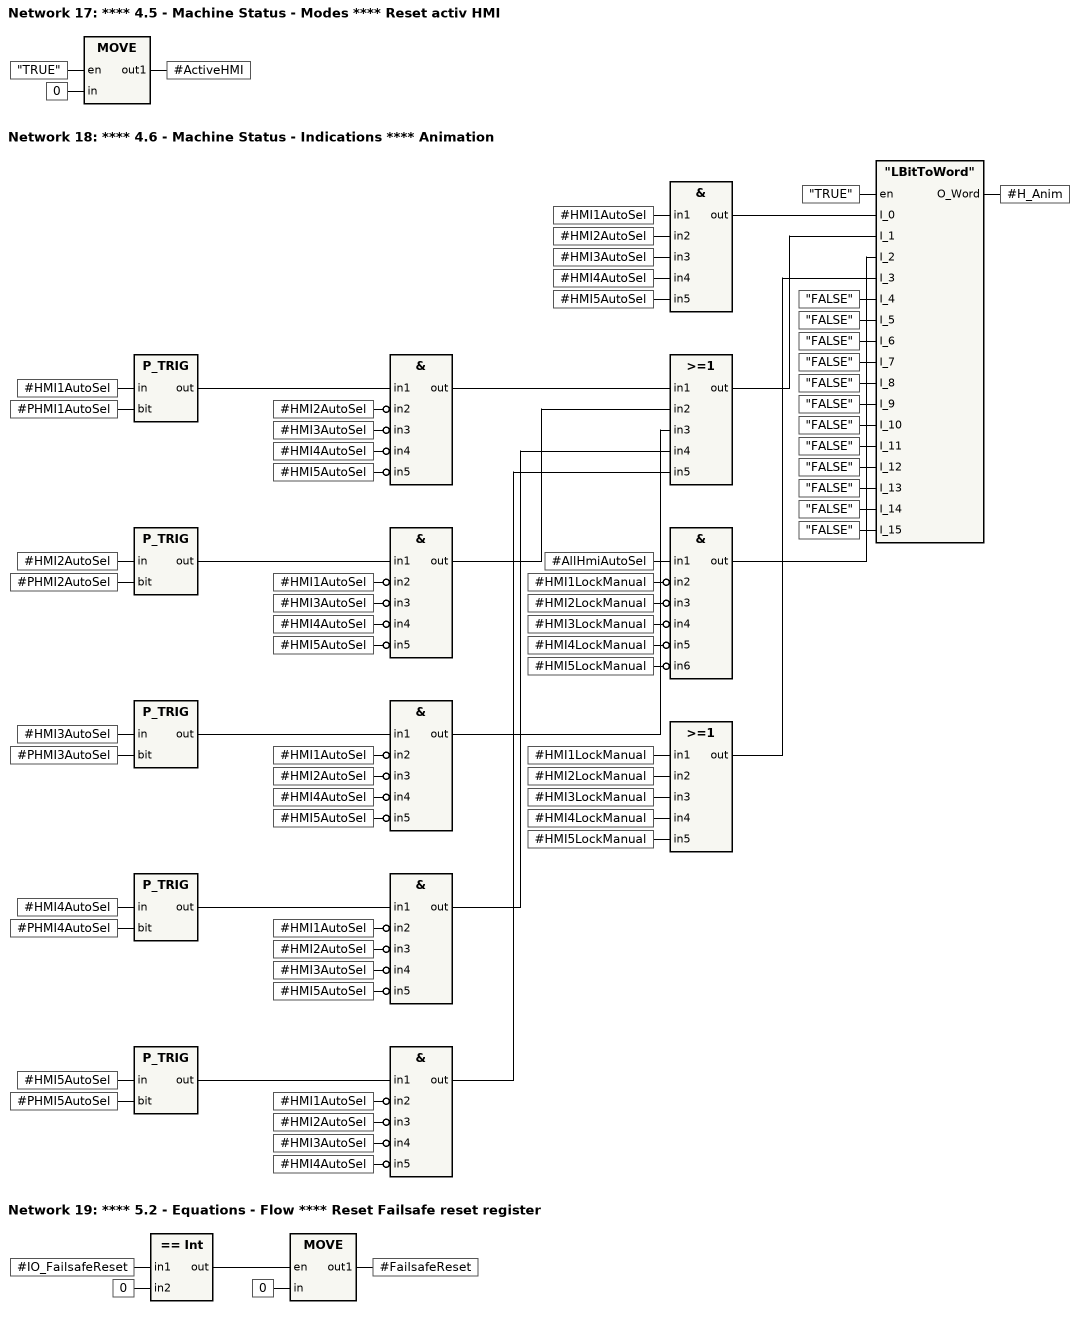
   IF "TRUE" THEN #ActiveHMI := 0; END_IF;
END_REGION

REGION Network 18: **** 4.6 - Machine Status - Indications **** Animation
   // Animation
   #_w1 := #HMI1AutoSel AND NOT #PHMI1AutoSel;   // rising edge
   #PHMI1AutoSel := #HMI1AutoSel;
   #_w2 := #HMI2AutoSel AND NOT #PHMI2AutoSel;   // rising edge
   #PHMI2AutoSel := #HMI2AutoSel;
   #_w3 := #HMI3AutoSel AND NOT #PHMI3AutoSel;   // rising edge
   #PHMI3AutoSel := #HMI3AutoSel;
   #_w4 := #HMI4AutoSel AND NOT #PHMI4AutoSel;   // rising edge
   #PHMI4AutoSel := #HMI4AutoSel;
   #_w5 := #HMI5AutoSel AND NOT #PHMI5AutoSel;   // rising edge
   #PHMI5AutoSel := #HMI5AutoSel;
   IF "TRUE" THEN
       "LBitToWord"(I_0 := #HMI1AutoSel AND #HMI2AutoSel AND #HMI3AutoSel AND #HMI4AutoSel AND #HMI5AutoSel,
                    I_1 := (#_w1 AND NOT #HMI2AutoSel AND NOT #HMI3AutoSel AND NOT #HMI4AutoSel AND NOT #HMI5AutoSel) OR (#_w2 AND NOT #HMI1AutoSel AND NOT #HMI3AutoSel AND NOT #HMI4AutoSel AND NOT #HMI5AutoSel) OR (#_w3 AND NOT #HMI1AutoSel AND NOT #HMI2AutoSel AND NOT #HMI4AutoSel AND NOT #HMI5AutoSel) OR (#_w4 AND NOT #HMI1AutoSel AND NOT #HMI2AutoSel AND NOT #HMI3AutoSel AND NOT #HMI5AutoSel) OR (#_w5 AND NOT #HMI1AutoSel AND NOT #HMI2AutoSel AND NOT #HMI3AutoSel AND NOT #HMI4AutoSel),
                    I_2 := #AllHmiAutoSel AND NOT #HMI1LockManual AND NOT #HMI2LockManual AND NOT #HMI3LockManual AND NOT #HMI4LockManual AND NOT #HMI5LockManual,
                    I_3 := #HMI1LockManual OR #HMI2LockManual OR #HMI3LockManual OR #HMI4LockManual OR #HMI5LockManual,
                    I_4 := "FALSE",
                    I_5 := "FALSE",
                    I_6 := "FALSE",
                    I_7 := "FALSE",
                    I_8 := "FALSE",
                    I_9 := "FALSE",
                    I_10 := "FALSE",
                    I_11 := "FALSE",
                    I_12 := "FALSE",
                    I_13 := "FALSE",
                    I_14 := "FALSE",
                    I_15 := "FALSE",
                    O_Word => #H_Anim);
   END_IF;
END_REGION

REGION Network 19: **** 5.2 - Equations - Flow **** Reset Failsafe reset register
   // Reset Failsafe reset register
   IF #IO_FailsafeReset = 0 THEN #FailsafeReset := 0; END_IF;
END_REGION

REGION Network 20: **** 5.2 - Equations - Flow **** Move 6 to the failsafe register when Alarm reset is slected on the HMI
   // Move 6 to the failsafe register when Alarm reset is slected on the HMI
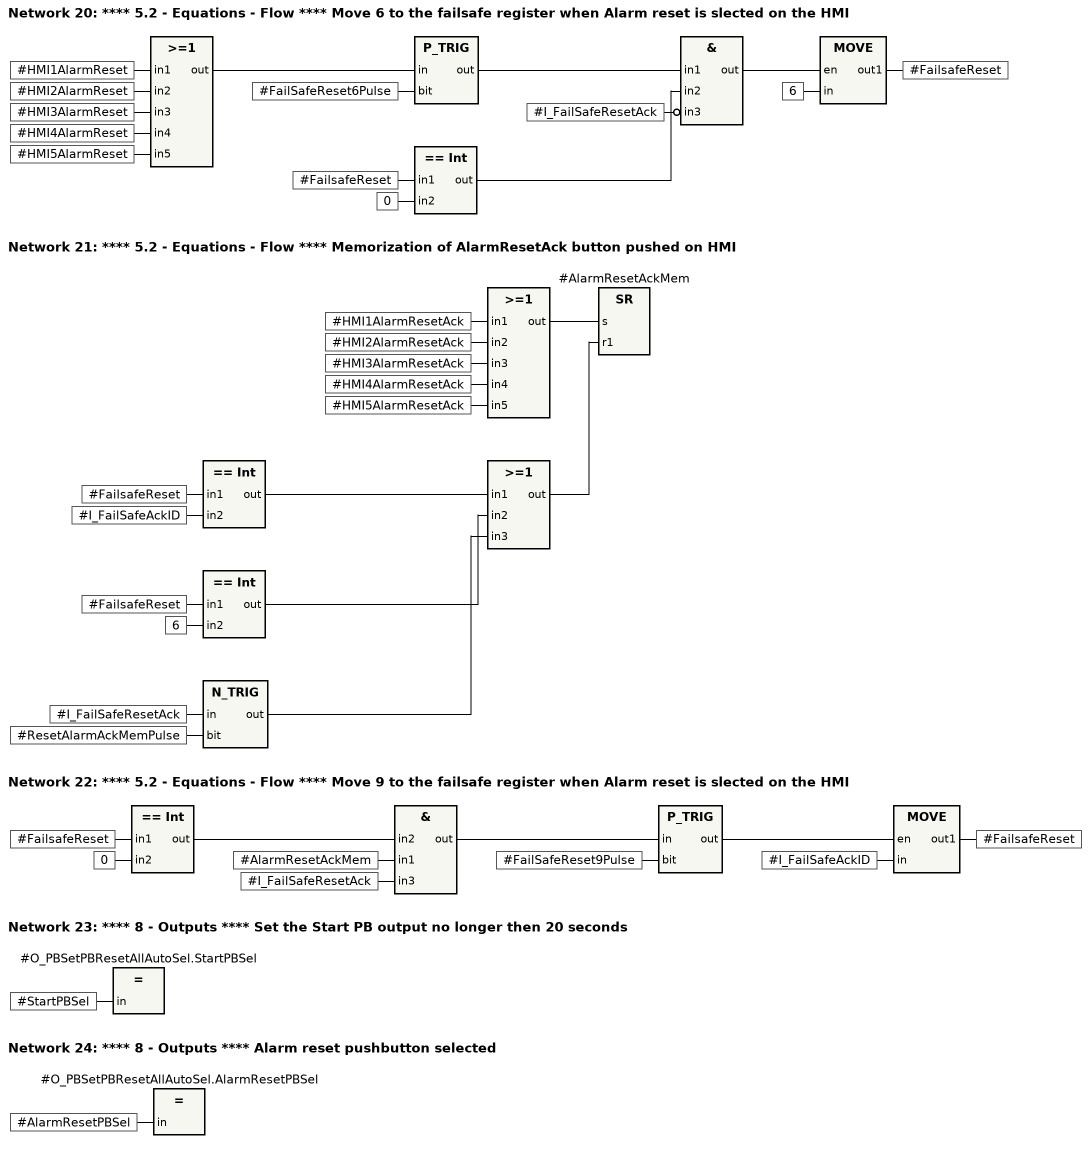
   #_w1 := #HMI1AlarmReset OR #HMI2AlarmReset OR #HMI3AlarmReset OR #HMI4AlarmReset OR #HMI5AlarmReset;
   #_w2 := #_w1 AND NOT #FailSafeReset6Pulse;   // rising edge
   #FailSafeReset6Pulse := #_w1;
   IF #_w2 AND (#FailsafeReset = 0) AND NOT #I_FailSafeResetAck THEN #FailsafeReset := 6; END_IF;
END_REGION

REGION Network 21: **** 5.2 - Equations - Flow **** Memorization of AlarmResetAck button pushed on HMI
   // Memorization of AlarmResetAck button pushed on HMI
   #_w1 := NOT #I_FailSafeResetAck AND #ResetAlarmAckMemPulse;   // falling edge
   #ResetAlarmAckMemPulse := #I_FailSafeResetAck;
   IF #HMI1AlarmResetAck OR #HMI2AlarmResetAck OR #HMI3AlarmResetAck OR #HMI4AlarmResetAck OR #HMI5AlarmResetAck THEN
       #AlarmResetAckMem := TRUE;   // SR flip-flop
   END_IF;
   IF (#FailsafeReset = #I_FailSafeAckID) OR (#FailsafeReset = 6) OR #_w1 THEN
       #AlarmResetAckMem := FALSE;
   END_IF;
END_REGION

REGION Network 22: **** 5.2 - Equations - Flow **** Move 9 to the failsafe register when Alarm reset is slected on the HMI
   // Move 9 to the failsafe register when Alarm reset is slected on the HMI
   #_w1 := (#FailsafeReset = 0) AND #AlarmResetAckMem AND #I_FailSafeResetAck;
   #_w2 := #_w1 AND NOT #FailSafeReset9Pulse;   // rising edge
   #FailSafeReset9Pulse := #_w1;
   IF #_w2 THEN #FailsafeReset := #I_FailSafeAckID; END_IF;
END_REGION

REGION Network 23: **** 8 - Outputs **** Set the Start PB output no longer then 20 seconds
   // Set the Start PB output no longer then 20 seconds
   #O_PBSetPBResetAllAutoSel.StartPBSel := #StartPBSel;
END_REGION

REGION Network 24: **** 8 - Outputs **** Alarm reset pushbutton selected
   // Alarm reset pushbutton selected
   #O_PBSetPBResetAllAutoSel.AlarmResetPBSel := #AlarmResetPBSel;
END_REGION

REGION Network 25: **** 8 - Outputs **** Set PB activated
   // Set PB activated
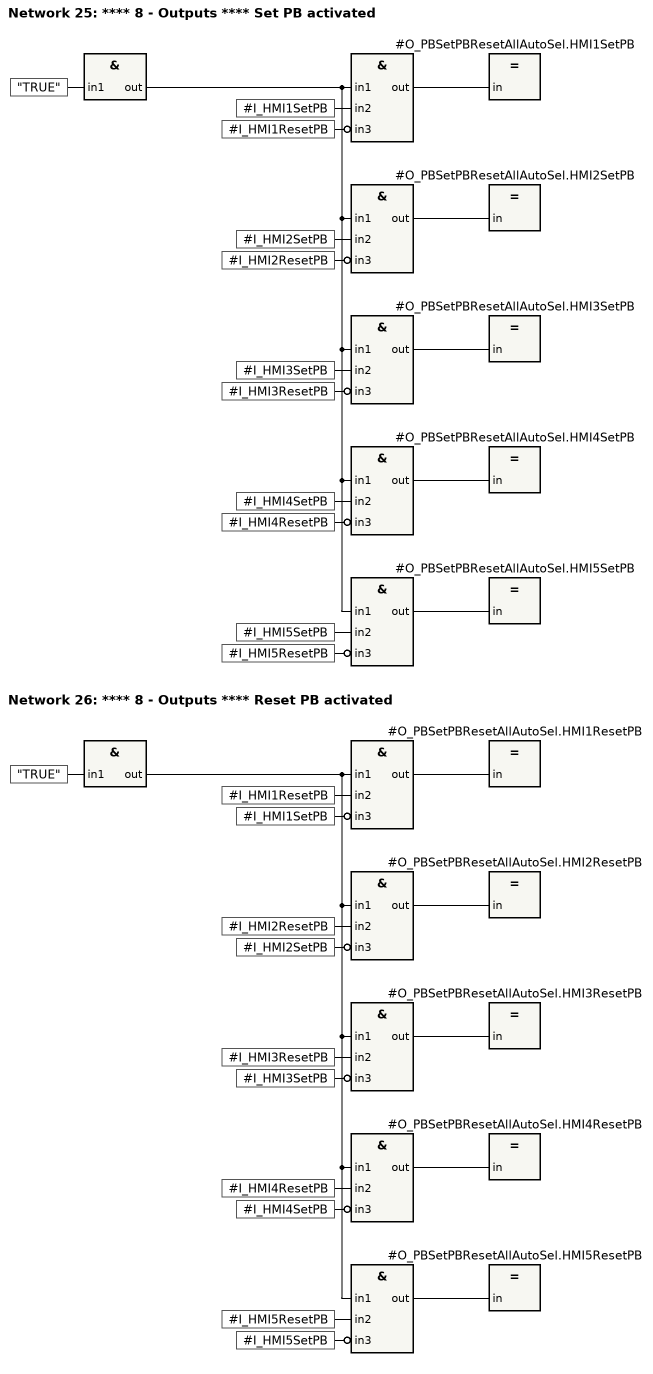
   #O_PBSetPBResetAllAutoSel.HMI1SetPB := "TRUE" AND #I_HMI1SetPB AND NOT #I_HMI1ResetPB;
   #O_PBSetPBResetAllAutoSel.HMI2SetPB := "TRUE" AND #I_HMI2SetPB AND NOT #I_HMI2ResetPB;
   #O_PBSetPBResetAllAutoSel.HMI3SetPB := "TRUE" AND #I_HMI3SetPB AND NOT #I_HMI3ResetPB;
   #O_PBSetPBResetAllAutoSel.HMI4SetPB := "TRUE" AND #I_HMI4SetPB AND NOT #I_HMI4ResetPB;
   #O_PBSetPBResetAllAutoSel.HMI5SetPB := "TRUE" AND #I_HMI5SetPB AND NOT #I_HMI5ResetPB;
END_REGION

REGION Network 26: **** 8 - Outputs **** Reset PB activated
   // Reset PB activated
   #O_PBSetPBResetAllAutoSel.HMI1ResetPB := "TRUE" AND #I_HMI1ResetPB AND NOT #I_HMI1SetPB;
   #O_PBSetPBResetAllAutoSel.HMI2ResetPB := "TRUE" AND #I_HMI2ResetPB AND NOT #I_HMI2SetPB;
   #O_PBSetPBResetAllAutoSel.HMI3ResetPB := "TRUE" AND #I_HMI3ResetPB AND NOT #I_HMI3SetPB;
   #O_PBSetPBResetAllAutoSel.HMI4ResetPB := "TRUE" AND #I_HMI4ResetPB AND NOT #I_HMI4SetPB;
   #O_PBSetPBResetAllAutoSel.HMI5ResetPB := "TRUE" AND #I_HMI5ResetPB AND NOT #I_HMI5SetPB;
END_REGION

REGION Network 27: **** 8 - Outputs **** All HMI Auto Sel
   // All HMI Auto Sel
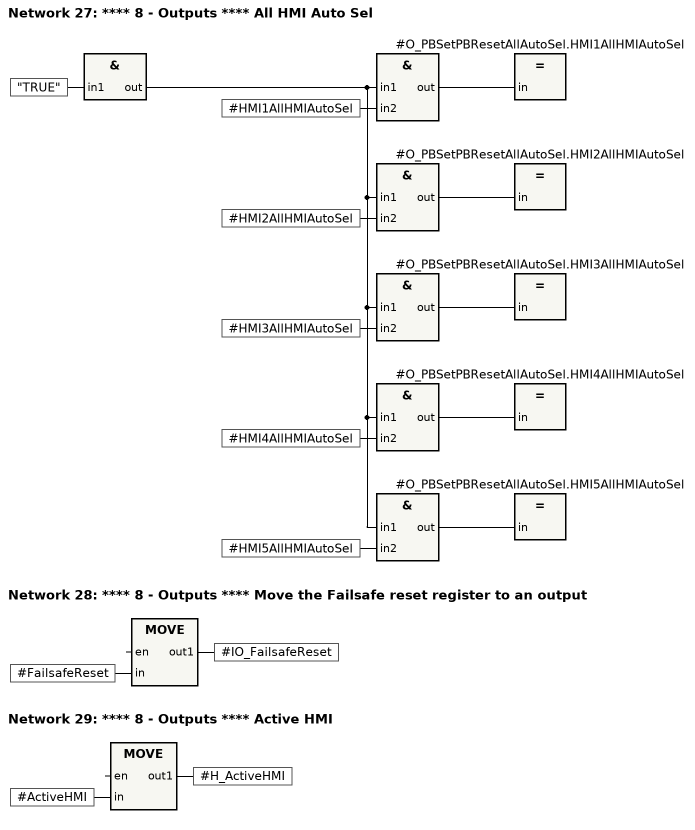
   #O_PBSetPBResetAllAutoSel.HMI1AllHMIAutoSel := "TRUE" AND #HMI1AllHMIAutoSel;
   #O_PBSetPBResetAllAutoSel.HMI2AllHMIAutoSel := "TRUE" AND #HMI2AllHMIAutoSel;
   #O_PBSetPBResetAllAutoSel.HMI3AllHMIAutoSel := "TRUE" AND #HMI3AllHMIAutoSel;
   #O_PBSetPBResetAllAutoSel.HMI4AllHMIAutoSel := "TRUE" AND #HMI4AllHMIAutoSel;
   #O_PBSetPBResetAllAutoSel.HMI5AllHMIAutoSel := "TRUE" AND #HMI5AllHMIAutoSel;
END_REGION

REGION Network 28: **** 8 - Outputs **** Move the Failsafe reset register to an output
   // Move the Failsafe reset register to an output
   #IO_FailsafeReset := #FailsafeReset;
END_REGION

REGION Network 29: **** 8 - Outputs **** Active HMI
   // Active HMI
   #H_ActiveHMI := #ActiveHMI;
END_REGION
END_FUNCTION_BLOCK

FUNCTION_BLOCK "LProcDO_NoFbk"   // FB1711, FBD
TITLE = LProcDO_NoFbk
{ S7_Optimized_Access := 'FALSE' }
AUTHOR : VCC
FAMILY : ProcEq
NAME : DONoFbk
VERSION : 0.1
// ================================================================================
// This module converts the signal 0-100% to digital commands Open and Close to 
// steer in position a valve or damper equipped with a motor.
// There is no feedback, the controller is operating with a time.
// Detections Open/Close may be connected to the controller to check the correct 
// opening and closing of the valve or damper.
// ================================================================================
// stored: AutoNumber false, IsIECCheckEnabled false, SetENOAutomatically False, UDAEnableTagReadback false
   VAR_INPUT
      I_CYCLE { ExternalAccessible := 'False'; ExternalVisible := 'False'; ExternalWritable := 'False'} : Time;   // Sample time
      H_PULSE_TM : Time;   // Minimum Pulse Time
      H_BREAK_TM : Time;   // Minimum Break Time
      H_MTR_TM : Time;   // Motor manipulated time value
      I_SP : Real;   // Set-point Input
      H_DEADB_W : Real;   // Slave: Deadband width
      I_COM_RST { ExternalAccessible := 'False'; ExternalVisible := 'False'; ExternalWritable := 'False'} : Bool;   // Initialising reset of controller
   END_VAR
   VAR_OUTPUT
      O_PosFbk { ExternalAccessible := 'False'; ExternalVisible := 'False'; ExternalWritable := 'False'} : Real;   // Output Feedback Position
      O_Set { ExternalAccessible := 'False'; ExternalVisible := 'False'; ExternalWritable := 'False'} : Bool;   // DO output Set
      O_Reset { ExternalAccessible := 'False'; ExternalVisible := 'False'; ExternalWritable := 'False'} : Bool;   // DO output Reset
   END_VAR
   VAR
      DO_Controller { ExternalAccessible := 'False'; ExternalVisible := 'False'; ExternalWritable := 'False'; S7_SetPoint := 'True'} : CONT_S;
   END_VAR
BEGIN

REGION Network 1: **** 5.2 - Equations - Flow Equations **** Activate DO controller
   // Activate DO controller
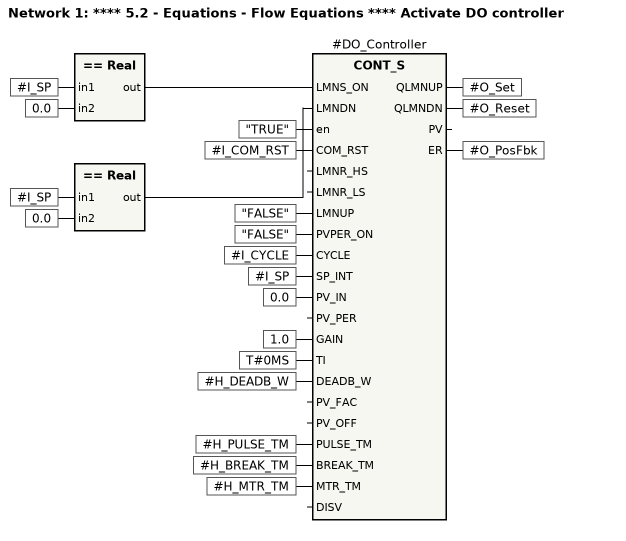
   IF "TRUE" THEN
       #DO_Controller(LMNS_ON := #I_SP = 0.0,   // CONT_S
                      LMNDN := #I_SP = 0.0,
                      COM_RST := #I_COM_RST,
                      LMNUP := "FALSE",
                      PVPER_ON := "FALSE",
                      CYCLE := #I_CYCLE,
                      SP_INT := #I_SP,
                      PV_IN := 0.0,
                      GAIN := 1.0,
                      TI := T#0MS,
                      DEADB_W := #H_DEADB_W,
                      PULSE_TM := #H_PULSE_TM,
                      BREAK_TM := #H_BREAK_TM,
                      MTR_TM := #H_MTR_TM,
                      QLMNUP => #O_Set,
                      QLMNDN => #O_Reset,
                      ER => #O_PosFbk);
   END_IF;
END_REGION
END_FUNCTION_BLOCK

FUNCTION_BLOCK "LProcSel5SP"   // FB1712, FBD
TITLE = LProcSel5SP
{ S7_Optimized_Access := 'FALSE' }
AUTHOR : VCC
FAMILY : ProcEq
NAME : Sel5SP
VERSION : 0.1
// ================================================================================
// This makes the selection of one set-point among 5 in function of the production 
// modes.
// The selection is made via a set-point request integer from 1 to 5.
// An external value is possible to be selected to set-point 1.
// ================================================================================
// stored: AutoNumber false, IsIECCheckEnabled false, SetENOAutomatically False, UDAEnableTagReadback false
   VAR_INPUT
      I_ExtSP1_Value { ExternalAccessible := 'False'; ExternalVisible := 'False'; ExternalWritable := 'False'} : Real;   // External Set-point 1
      H_SP2 : Real;   // Set-point 2
      H_SP3 : Real;   // Set-point 3
      H_SP4 : Real;   // Set-point 4
      H_SP5 : Real;   // Set-point 5
      I_SPReq : Int;   // Index Set-point Request
      I_ExtSP1 : Bool;   // External Set-point 1 Request
   END_VAR
   VAR_OUTPUT
      O_SPSel : Real;   // Set-point selected
   END_VAR
   VAR_IN_OUT
      H_SP1 : Real;   // Set-point 1
   END_VAR
BEGIN

REGION Network 1: **** 5.2 - Equations - Flow Equations **** Selection Set-point 1
   // Selection Set-point 1
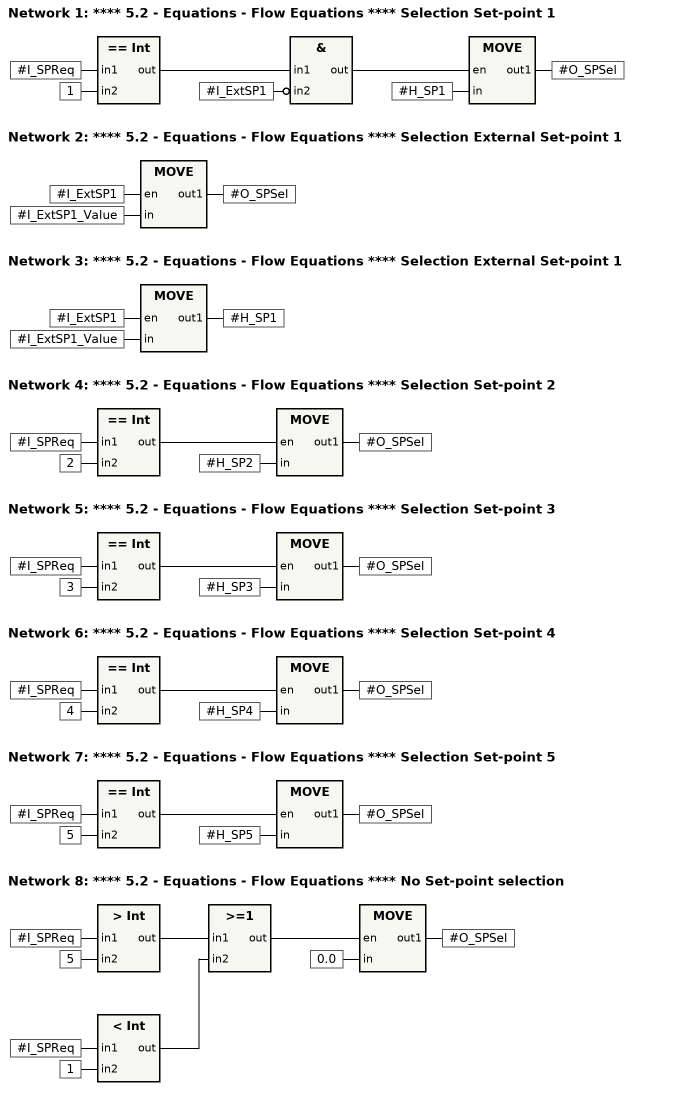
   IF (#I_SPReq = 1) AND NOT #I_ExtSP1 THEN #O_SPSel := #H_SP1; END_IF;
END_REGION

REGION Network 2: **** 5.2 - Equations - Flow Equations **** Selection External Set-point 1
   // Selection External Set-point 1
   IF #I_ExtSP1 THEN #O_SPSel := #I_ExtSP1_Value; END_IF;
END_REGION

REGION Network 3: **** 5.2 - Equations - Flow Equations **** Selection External Set-point 1
   // Selection External Set-point 1
   IF #I_ExtSP1 THEN #H_SP1 := #I_ExtSP1_Value; END_IF;
END_REGION

REGION Network 4: **** 5.2 - Equations - Flow Equations **** Selection Set-point 2
   // Selection Set-point 2
   IF #I_SPReq = 2 THEN #O_SPSel := #H_SP2; END_IF;
END_REGION

REGION Network 5: **** 5.2 - Equations - Flow Equations **** Selection Set-point 3
   // Selection Set-point 3
   IF #I_SPReq = 3 THEN #O_SPSel := #H_SP3; END_IF;
END_REGION

REGION Network 6: **** 5.2 - Equations - Flow Equations **** Selection Set-point 4
   // Selection Set-point 4
   IF #I_SPReq = 4 THEN #O_SPSel := #H_SP4; END_IF;
END_REGION

REGION Network 7: **** 5.2 - Equations - Flow Equations **** Selection Set-point 5
   // Selection Set-point 5
   IF #I_SPReq = 5 THEN #O_SPSel := #H_SP5; END_IF;
END_REGION

REGION Network 8: **** 5.2 - Equations - Flow Equations **** No Set-point selection
   // No Set-point selection
   IF (#I_SPReq > 5) OR (#I_SPReq < 1) THEN #O_SPSel := 0.0; END_IF;
END_REGION
END_FUNCTION_BLOCK

FUNCTION_BLOCK "LProcPid"   // FB1713, FBD
TITLE = LProcPid
{ S7_Optimized_Access := 'FALSE' }
AUTHOR : VCC
FAMILY : ProcEq
NAME : Pid
VERSION : 0.1
// ================================================================================
// The Process Value is controlled by the Pid controller.
// ================================================================================
// stored: AutoNumber false, IsIECCheckEnabled false, SetENOAutomatically False, UDAEnableTagReadback false
   VAR_INPUT
      I_CYCLE { ExternalAccessible := 'False'; ExternalVisible := 'False'; ExternalWritable := 'False'} : Time;   // Sample time
      H_TI : Time;   // Pid Reset time
      H_TD : Time;   // Pid Derivative time
      I_Manual_Value { ExternalAccessible := 'False'; ExternalVisible := 'False'; ExternalWritable := 'False'} : Real;   // Pid Setpoint Manual
      I_SP_Auto : Real;   // Pid Setpoint for controller
      I_PV_PID : Real;   // Pid Process value
      H_GAIN : Real;   // Pid Proportional Gain
      H_DEADB_W : Real;   // Pid Deadband width
      H_LMN_HLM : Real := 100.0;   // Pid Manipulated value high limit
      H_LMN_LLM : Real;   // Pid Manipulated value low limit
      I_COM_RST { ExternalAccessible := 'False'; ExternalVisible := 'False'; ExternalWritable := 'False'} : Bool;   // Initialising reset of controller
      I_MAN_ON { ExternalAccessible := 'False'; ExternalVisible := 'False'; ExternalWritable := 'False'} : Bool;   // Pid Manual value on
      H_Direct : Bool := TRUE;   // Pid in Direct mode (output increase if SP>PV)
      H_P_SEL : Bool;   // Pid P selected
      H_I_SEL : Bool;   // Pid I selected
      H_D_SEL : Bool;   // Pid D selected
   END_VAR
   VAR_OUTPUT
      O_SP_PID : Real;   // Setpoint used in Pid controller
      O_LMN_PID : Real;   // Output value Pid Controller
   END_VAR
   VAR DB_SPECIFIC
      Gain { ExternalAccessible := 'False'; ExternalVisible := 'False'; ExternalWritable := 'False'} : Real;   // Pid Gain in function of Pid direct or not
      DirectCoef { ExternalAccessible := 'False'; ExternalVisible := 'False'; ExternalWritable := 'False'} : Real;   // Value +1 or -1 if Pid direct or not
      M_LMN { ExternalAccessible := 'False'; ExternalVisible := 'False'; ExternalWritable := 'False'} : Real;   // Pid Manipulated value from controller
   END_VAR
   VAR
      PidControl { ExternalAccessible := 'False'; ExternalVisible := 'False'; ExternalWritable := 'False'; S7_SetPoint := 'True'} : CONT_C;   // Pid Controller
   END_VAR
BEGIN

REGION Network 1: **** 7 - Submodules - Non-machine **** Pid control Direct: Gain>0 and Output increase when SP>PV
   // Pid control Direct: Gain>0 and Output increase when SP>PV
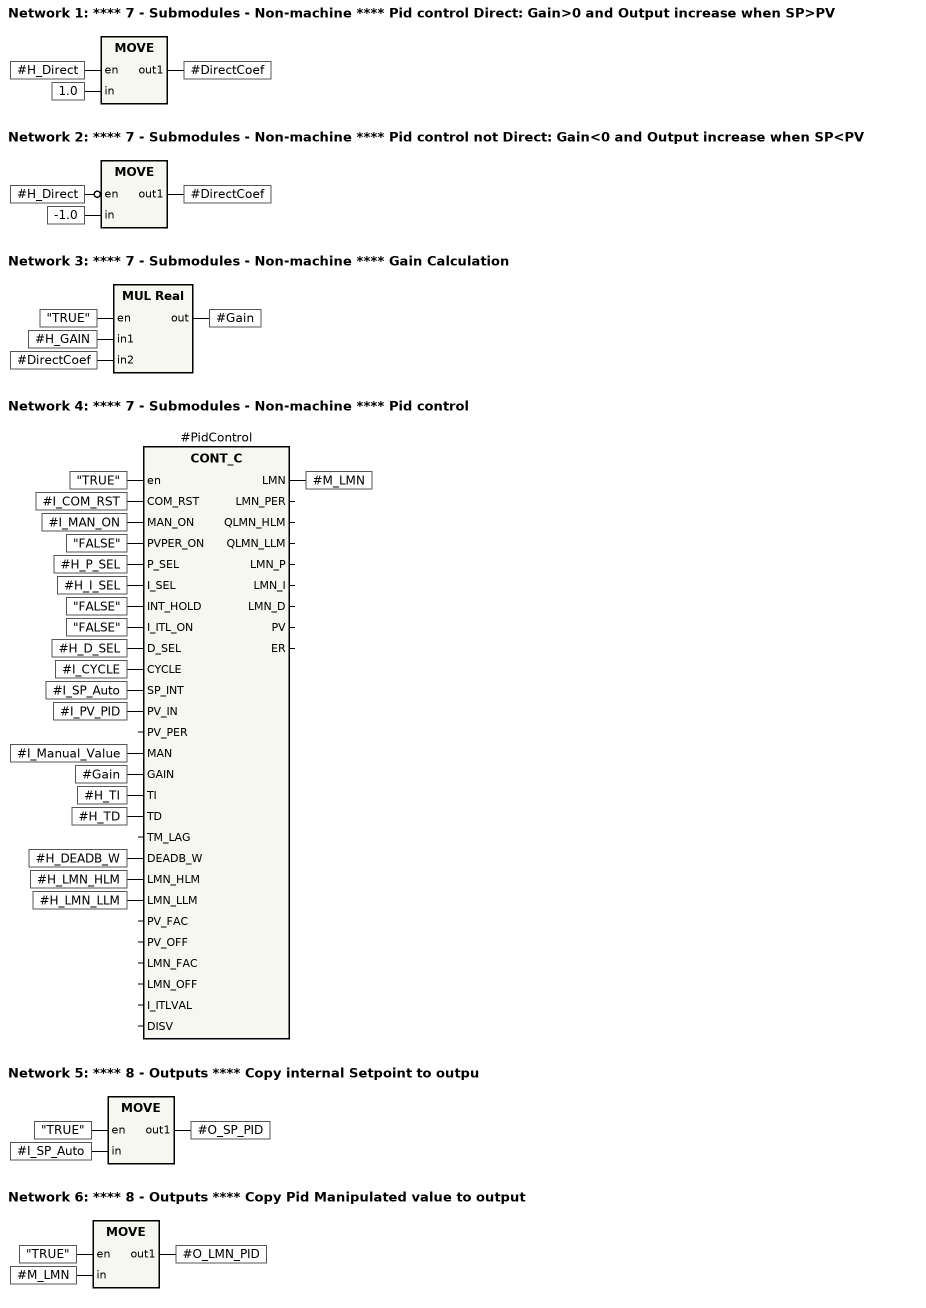
   IF #H_Direct THEN #DirectCoef := 1.0; END_IF;
END_REGION

REGION Network 2: **** 7 - Submodules - Non-machine **** Pid control not Direct: Gain<0 and Output increase when SP<PV
   // Pid control not Direct: Gain<0 and Output increase when SP<PV
   IF NOT #H_Direct THEN #DirectCoef := -1.0; END_IF;
END_REGION

REGION Network 3: **** 7 - Submodules - Non-machine **** Gain Calculation
   // Gain Calculation
   IF "TRUE" THEN #Gain := #H_GAIN * #DirectCoef; END_IF;
END_REGION

REGION Network 4: **** 7 - Submodules - Non-machine **** Pid control
   // Pid control
   IF "TRUE" THEN
       #PidControl(COM_RST := #I_COM_RST,   // CONT_C
                   MAN_ON := #I_MAN_ON,
                   PVPER_ON := "FALSE",
                   P_SEL := #H_P_SEL,
                   I_SEL := #H_I_SEL,
                   INT_HOLD := "FALSE",
                   I_ITL_ON := "FALSE",
                   D_SEL := #H_D_SEL,
                   CYCLE := #I_CYCLE,
                   SP_INT := #I_SP_Auto,
                   PV_IN := #I_PV_PID,
                   MAN := #I_Manual_Value,
                   GAIN := #Gain,
                   TI := #H_TI,
                   TD := #H_TD,
                   DEADB_W := #H_DEADB_W,
                   LMN_HLM := #H_LMN_HLM,
                   LMN_LLM := #H_LMN_LLM,
                   LMN => #M_LMN);
   END_IF;
END_REGION

REGION Network 5: **** 8 - Outputs **** Copy internal Setpoint to outpu
   // Copy internal Setpoint to output
   IF "TRUE" THEN #O_SP_PID := #I_SP_Auto; END_IF;
END_REGION

REGION Network 6: **** 8 - Outputs **** Copy Pid Manipulated value to output
   // Copy Pid Manipulated value to output
   IF "TRUE" THEN #O_LMN_PID := #M_LMN; END_IF;
END_REGION
END_FUNCTION_BLOCK

FUNCTION_BLOCK "LProcMotor1W1S-S"   // FB1714, FBD
TITLE = LProcMotor1W1S-S
{ S7_Optimized_Access := 'FALSE' }
AUTHOR : VCC
FAMILY : ProcEq
NAME : M1W1S-S
VERSION : 0.6
// ===============================================================================
// This "Motor-1Way-1Speed-SoftStarter" module is used in applications when a 
// motor 1 way - 1 speed equipped with SoftStarter is needed.
// The module contains: a motor loop equipped with 
// "1 mode from HMI
// "1 motor protection.
// "1 safety switch.
// "1 feedback motor running (option): Pressure-switch, Rotation guard,........
// "1 bypass contactor.
// "1 bypass key-switch.
// "1 softstarter.
// ===============================================================================
// stored: AutoNumber false, IsIECCheckEnabled false, SetENOAutomatically False, UDAEnableTagReadback false
   VAR_INPUT
      I_RunFbkAlarmTime { ExternalAccessible := 'False'; ExternalVisible := 'False'; ExternalWritable := 'False'} : DInt;   // Time for alarm Feedback Motor running
      I_EnableAlarm { ExternalAccessible := 'False'; ExternalVisible := 'False'; ExternalWritable := 'False'} : Bool;   // Enable alarm
      I_AutoReq { ExternalAccessible := 'False'; ExternalVisible := 'False'; ExternalWritable := 'False'} : Bool;   // Auto Request from equation or Sequence
      I_InterlockOk { ExternalAccessible := 'False'; ExternalVisible := 'False'; ExternalWritable := 'False'} : Bool;   // Interlock Ok
      I_MotorProtection { ExternalAccessible := 'False'; ExternalVisible := 'False'; ExternalWritable := 'False'} : Bool;   // Motor protection Ok
      I_SoftStarterOK { ExternalAccessible := 'False'; ExternalVisible := 'False'; ExternalWritable := 'False'} : Bool;   // SoftStarter Ok
      I_EndOfRamp { ExternalAccessible := 'False'; ExternalVisible := 'False'; ExternalWritable := 'False'} : Bool;   // SoftStarter End Of Ramp
      I_BypassKey { ExternalAccessible := 'False'; ExternalVisible := 'False'; ExternalWritable := 'False'} : Bool;   // Bypass Key-switch
      I_SafetySwitch { ExternalAccessible := 'False'; ExternalVisible := 'False'; ExternalWritable := 'False'} : Bool;   // Safety Switch Ok
      I_RunFeedBack { ExternalAccessible := 'False'; ExternalVisible := 'False'; ExternalWritable := 'False'} : Bool;   // Feedback motor running (Pressure-switch, Rotation Guard,...)
      I_PBSetPBResetAllAutoSel { ExternalAccessible := 'False'; ExternalVisible := 'False'; ExternalWritable := 'False'} : Struct   // Set PB activated - Reset PB activated - All HMI Auto selected
         HMI1SetPB { ExternalAccessible := 'False'; ExternalVisible := 'False'; ExternalWritable := 'False'} : Bool;   // Set PB activated on HMI1
         HMI1ResetPB { ExternalAccessible := 'False'; ExternalVisible := 'False'; ExternalWritable := 'False'} : Bool;   // Reset PB activated on HMI1
         HMI1AllHMIAutoSel { ExternalAccessible := 'False'; ExternalVisible := 'False'; ExternalWritable := 'False'} : Bool;   // All HMI Auto selected on HMI1
         HMI2SetPB { ExternalAccessible := 'False'; ExternalVisible := 'False'; ExternalWritable := 'False'} : Bool;   // Set PB activated on HMI2
         HMI2ResetPB { ExternalAccessible := 'False'; ExternalVisible := 'False'; ExternalWritable := 'False'} : Bool;   // Reset PB activated on HMI2
         HMI2AllHMIAutoSel { ExternalAccessible := 'False'; ExternalVisible := 'False'; ExternalWritable := 'False'} : Bool;   // All HMI Auto selected on HMI2
         HMI3SetPB { ExternalAccessible := 'False'; ExternalVisible := 'False'; ExternalWritable := 'False'} : Bool;   // Set PB activated on HMI3
         HMI3ResetPB { ExternalAccessible := 'False'; ExternalVisible := 'False'; ExternalWritable := 'False'} : Bool;   // Reset PB activated on HMI3
         HMI3AllHMIAutoSel { ExternalAccessible := 'False'; ExternalVisible := 'False'; ExternalWritable := 'False'} : Bool;   // All HMI Auto selected on HMI3
         HMI4SetPB { ExternalAccessible := 'False'; ExternalVisible := 'False'; ExternalWritable := 'False'} : Bool;   // Set PB activated on HMI4
         HMI4ResetPB { ExternalAccessible := 'False'; ExternalVisible := 'False'; ExternalWritable := 'False'} : Bool;   // Reset PB activated on HMI4
         HMI4AllHMIAutoSel { ExternalAccessible := 'False'; ExternalVisible := 'False'; ExternalWritable := 'False'} : Bool;   // All HMI Auto selected on HMI4
         HMI5SetPB { ExternalAccessible := 'False'; ExternalVisible := 'False'; ExternalWritable := 'False'} : Bool;   // Set PB activated on HMI5
         HMI5ResetPB { ExternalAccessible := 'False'; ExternalVisible := 'False'; ExternalWritable := 'False'} : Bool;   // Reset PB activated on HMI5
         HMI5AllHMIAutoSel { ExternalAccessible := 'False'; ExternalVisible := 'False'; ExternalWritable := 'False'} : Bool;   // All HMI Auto selected on HMI5
         StartPBSel { ExternalAccessible := 'False'; ExternalVisible := 'False'; ExternalWritable := 'False'} : Bool;   // Start is activated
         AlarmResetPBSel { ExternalAccessible := 'False'; ExternalVisible := 'False'; ExternalWritable := 'False'} : Bool;   // Alarm reset is activated
      END_STRUCT;
      I_UpperLevelAlarmA { ExternalAccessible := 'False'; ExternalVisible := 'False'; ExternalWritable := 'False'} : Bool;   // Upper level alarm A
      I_UpperLevelAlarmB { ExternalAccessible := 'False'; ExternalVisible := 'False'; ExternalWritable := 'False'} : Bool;   // Upper level alarm B
      C_EnableSetResetHMI { ExternalAccessible := 'False'; ExternalVisible := 'False'; ExternalWritable := 'False'} : Bool;   // Enable Set-Reset functions from HMI
      C_SelfHolding { ExternalAccessible := 'False'; ExternalVisible := 'False'; ExternalWritable := 'False'} : Bool := TRUE;   // Enable SelfHolding Command
      C_RunFeedBackUsed { ExternalAccessible := 'False'; ExternalVisible := 'False'; ExternalWritable := 'False'} : Bool;   // Feedback motor running is used
      C_SafetySwNc { ExternalAccessible := 'False'; ExternalVisible := 'False'; ExternalWritable := 'False'} : Bool;   // Safety switch Normally closed
      C_MotorProtectionNc { ExternalAccessible := 'False'; ExternalVisible := 'False'; ExternalWritable := 'False'} : Bool;   // Motor protection Normally closed
      C_BypassSw_HW { ExternalAccessible := 'False'; ExternalVisible := 'False'; ExternalWritable := 'False'} : Bool := TRUE;   // Bypass-switch Hardware (=true) otherwise Software
      C_BypassSwOffFault { ExternalAccessible := 'False'; ExternalVisible := 'False'; ExternalWritable := 'False'} : Bool := TRUE;   // Bypass Switch active when input = False
      C_ManualForced { ExternalAccessible := 'False'; ExternalVisible := 'False'; ExternalWritable := 'False'} : Bool;   // Manual Forced is used (=true)
   END_VAR
   VAR_OUTPUT
      O_Contactor { ExternalAccessible := 'False'; ExternalVisible := 'False'; ExternalWritable := 'False'} : Bool;   // Bypass Contactor of motor loop
      O_Start { ExternalAccessible := 'False'; ExternalVisible := 'False'; ExternalWritable := 'False'} : Bool;   // Start Command SoftStarter
      O_AlarmA { ExternalAccessible := 'False'; ExternalVisible := 'False'; ExternalWritable := 'False'} : Bool;   // Alarm A
      O_AlarmB { ExternalAccessible := 'False'; ExternalVisible := 'False'; ExternalWritable := 'False'} : Bool;   // Alarm B
      O_AlarmC { ExternalAccessible := 'False'; ExternalVisible := 'False'; ExternalWritable := 'False'} : Bool;   // Alarm C
      O_AlarmD { ExternalAccessible := 'False'; ExternalVisible := 'False'; ExternalWritable := 'False'} : Bool;   // Alarm D
      O_AlarmABCondition { ExternalAccessible := 'False'; ExternalVisible := 'False'; ExternalWritable := 'False'} : Bool;   // Alarms resetable
      H_IAnim { ExternalAccessible := 'False'; ExternalVisible := 'False'; ExternalWritable := 'False'} : Word;   // HMI Animation color of the icon
      H_AlarmWord { ExternalAccessible := 'False'; ExternalVisible := 'False'; ExternalWritable := 'False'} : DWord;   // Alarm Word
   END_VAR
   VAR DB_SPECIFIC
      AA_SafetySwitch { ExternalAccessible := 'False'; ExternalVisible := 'False'; ExternalWritable := 'False'} : Bool;   // Safety Switch alarm
      AA_MotorProtection { ExternalAccessible := 'False'; ExternalVisible := 'False'; ExternalWritable := 'False'} : Bool;   // Motor Protection alarm
      AA_SoftStarter { ExternalAccessible := 'False'; ExternalVisible := 'False'; ExternalWritable := 'False'} : Bool;   // SoftStarter Alarm
      AB_RunFeedback { ExternalAccessible := 'False'; ExternalVisible := 'False'; ExternalWritable := 'False'} : Bool;   // Motor Running Feedback Alarm
      AB_OvTimeAutoSel { ExternalAccessible := 'False'; ExternalVisible := 'False'; ExternalWritable := 'False'} : Bool;   // Overtime Auto selected
      AD_BypassSwitch { ExternalAccessible := 'False'; ExternalVisible := 'False'; ExternalWritable := 'False'} : Bool;   // Bypass-Switch Alarm
      AD_BypassSoftKey { ExternalAccessible := 'False'; ExternalVisible := 'False'; ExternalWritable := 'False'} : Bool;   // Bypass-Key HMI Alarm
      AD_InterlockAlarm { ExternalAccessible := 'False'; ExternalVisible := 'False'; ExternalWritable := 'False'} : Bool;   // Interlock Fault
      H_HMIModeCmd : Word;   // Mode commands from HMI
      H_ActiveHMI : Int;   // Active HMI
      H_NameActiveHMI : String[25];   // Name of the Active HMI
      H_Out : Struct   // HMI
         MotorProtectIAnim : Word;   // HMI Animation color of object
         SafetySwitchIAnim : Word;   // HMI Animation color of object
         SoftStarterIAnim : Word;   // HMI Animation color of object
         StartRelayIAnim : Word;   // HMI Animation color of object
         ContactorIAnim : Word;   // HMI Animation color of object
         BypassSwitchIAnim : Word;   // HMI Animation color of object
         RunFbkIAnim : Word;   // HMI Animation color of object
         Anim : Word;   // HMI Animation word
         Anim2 : Word;   // HMI Animation word
         Anim3 : Bool;   // HMI Animation bool
         DBnr : Int;   // HMI Animation DB number
      END_STRUCT;
      AutoMode { ExternalAccessible := 'False'; ExternalVisible := 'False'; ExternalWritable := 'False'} : Bool;   // Auto mode
      ManualMode { ExternalAccessible := 'False'; ExternalVisible := 'False'; ExternalWritable := 'False'} : Bool;   // Manual mode
      AutoModeSel { ExternalAccessible := 'False'; ExternalVisible := 'False'; ExternalWritable := 'False'} : Bool;   // Auto Mode Selection from HMI
      ManualModeSel { ExternalAccessible := 'False'; ExternalVisible := 'False'; ExternalWritable := 'False'} : Bool;   // Manual Mode Selection from HMI
      HMISetCmd { ExternalAccessible := 'False'; ExternalVisible := 'False'; ExternalWritable := 'False'} : Bool;   // Set Command on HMI
      HMIResetCmd { ExternalAccessible := 'False'; ExternalVisible := 'False'; ExternalWritable := 'False'} : Bool;   // Reset Command on HMI
      H_FncSelInHMI { ExternalAccessible := 'False'; ExternalVisible := 'False'; ExternalWritable := 'False'} : Bool;   // Manual selection from HMI
      ForcedMan { ExternalAccessible := 'False'; ExternalVisible := 'False'; ExternalWritable := 'False'} : Bool;   // Forced manual active
      ForcedManTimer { ExternalAccessible := 'False'; ExternalVisible := 'False'; ExternalWritable := 'False'} : Bool;   // Forced manual timer
      OvTimeAutoSel { ExternalAccessible := 'False'; ExternalVisible := 'False'; ExternalWritable := 'False'} : Bool;   // Overtime Auto selected
      OvTimeAutoSelCond { ExternalAccessible := 'False'; ExternalVisible := 'False'; ExternalWritable := 'False'} : Bool;   // Overtime Auto selected condition
      MotorProtectionABCond { ExternalAccessible := 'False'; ExternalVisible := 'False'; ExternalWritable := 'False'} : Bool;   // Motor protection alarm can be reset
      MotorProtectionAlm { ExternalAccessible := 'False'; ExternalVisible := 'False'; ExternalWritable := 'False'} : Bool;   // Motor protection alarm
      MotorProtectionDisable { ExternalAccessible := 'False'; ExternalVisible := 'False'; ExternalWritable := 'False'} : Bool;   // Motor protection alarm is disabled from HMI
      SafetySwitchABCond { ExternalAccessible := 'False'; ExternalVisible := 'False'; ExternalWritable := 'False'} : Bool;   // Safety Switch alarm can be reset
      SafetySwitchAlm { ExternalAccessible := 'False'; ExternalVisible := 'False'; ExternalWritable := 'False'} : Bool;   // Safety Switch alarm
      SafetySwitchDisable { ExternalAccessible := 'False'; ExternalVisible := 'False'; ExternalWritable := 'False'} : Bool;   // Safety Switch alarm is disabled from HMI
      SoftStarterABCond { ExternalAccessible := 'False'; ExternalVisible := 'False'; ExternalWritable := 'False'} : Bool;   // SoftStarter alarm can be reset
      SoftStarterDisable { ExternalAccessible := 'False'; ExternalVisible := 'False'; ExternalWritable := 'False'} : Bool;   // SoftStarter alarm is disabled from HMI
      BypassSwitchDisable { ExternalAccessible := 'False'; ExternalVisible := 'False'; ExternalWritable := 'False'} : Bool;   // Bypass-switch alarm is disabled from HMI
      BypassForced { ExternalAccessible := 'False'; ExternalVisible := 'False'; ExternalWritable := 'False'} : Bool;   // Bypass Forced by Key-switch
      RunFbkEnAlarm { ExternalAccessible := 'False'; ExternalVisible := 'False'; ExternalWritable := 'False'} : Bool;   // Motor Running Feedback Enable Alarm
      RunFbkDisable { ExternalAccessible := 'False'; ExternalVisible := 'False'; ExternalWritable := 'False'} : Bool;   // Motor Running Feedback Alarm is disabled from HMI
      RunFeedBackABCond { ExternalAccessible := 'False'; ExternalVisible := 'False'; ExternalWritable := 'False'} : Bool;   // Motor Running Feedback Alarm can be reset
      CmdRequest { ExternalAccessible := 'False'; ExternalVisible := 'False'; ExternalWritable := 'False'} : Bool;   // Command request to activate the component
      SetPBMan { ExternalAccessible := 'False'; ExternalVisible := 'False'; ExternalWritable := 'False'} : Bool;   // Set pushbutton is activated in manual
      ResetPBMan { ExternalAccessible := 'False'; ExternalVisible := 'False'; ExternalWritable := 'False'} : Bool;   // Reset pushbutton is activated in manual
      AllHMIAutoSel { ExternalAccessible := 'False'; ExternalVisible := 'False'; ExternalWritable := 'False'} : Bool;   // All HMI Auto selected
      Active { ExternalAccessible := 'False'; ExternalVisible := 'False'; ExternalWritable := 'False'} : Bool;   // Motor Loop is active
      Contactor { ExternalAccessible := 'False'; ExternalVisible := 'False'; ExternalWritable := 'False'} : Bool;   // Contactor
      StartCmd { ExternalAccessible := 'False'; ExternalVisible := 'False'; ExternalWritable := 'False'} : Bool;   // Start Command
      AlarmA { ExternalAccessible := 'False'; ExternalVisible := 'False'; ExternalWritable := 'False'} : Bool;   // Summation Alarm A
      AlarmB { ExternalAccessible := 'False'; ExternalVisible := 'False'; ExternalWritable := 'False'} : Bool;   // Summation Alarm B
      AlarmC { ExternalAccessible := 'False'; ExternalVisible := 'False'; ExternalWritable := 'False'} : Bool;   // Summation Alarm C
      AlarmD { ExternalAccessible := 'False'; ExternalVisible := 'False'; ExternalWritable := 'False'} : Bool;   // Summation Alarm D
      DBnr { ExternalAccessible := 'False'; ExternalVisible := 'False'; ExternalWritable := 'False'} : Int;   // HMI DB number
   END_VAR
   VAR
      TimerForcedMan { ExternalAccessible := 'False'; ExternalVisible := 'False'; ExternalWritable := 'False'; S7_SetPoint := 'True'} : "LTimer";   // Timer Manual Forced
      OvtAutoSelTimer { ExternalAccessible := 'False'; ExternalVisible := 'False'; ExternalWritable := 'False'; S7_SetPoint := 'True'} : "LTimer";   // Timer Overtime Auto Selection
      RunFbkTimer { ExternalAccessible := 'False'; ExternalVisible := 'False'; ExternalWritable := 'False'; S7_SetPoint := 'True'} : "LTimer";   // Timer Run Feedback Alarm
      RunFeedback { ExternalAccessible := 'False'; ExternalVisible := 'False'; ExternalWritable := 'False'; S7_SetPoint := 'True'} : "LProc1AlarmMultiIn";   // Run Feedback Alarm
      MotorProtection { ExternalAccessible := 'False'; ExternalVisible := 'False'; ExternalWritable := 'False'; S7_SetPoint := 'True'} : "LProc1AlarmMultiIn";   // Motor protection alarm
      SafetySwitch { ExternalAccessible := 'False'; ExternalVisible := 'False'; ExternalWritable := 'False'; S7_SetPoint := 'True'} : "LProc1AlarmMultiIn";   // Safety Switch alarm
      SoftStarter { ExternalAccessible := 'False'; ExternalVisible := 'False'; ExternalWritable := 'False'; S7_SetPoint := 'True'} : "LProc1AlarmMultiIn";   // SoftStarter alarm
      BypassSwitch { ExternalAccessible := 'False'; ExternalVisible := 'False'; ExternalWritable := 'False'; S7_SetPoint := 'True'} : "LProc1AlarmMultiIn";   // Bypass alarm
      Modes { ExternalAccessible := 'False'; ExternalVisible := 'False'; ExternalWritable := 'False'; S7_SetPoint := 'True'} : "LProcObjectMode";
   END_VAR
   VAR DB_SPECIFIC
      CheckActiveHMI { ExternalAccessible := 'False'; ExternalVisible := 'False'; ExternalWritable := 'False'; S7_SetPoint := 'True'} : TP_TIME;   // Timer
      CheckActiveHMI_1 { ExternalAccessible := 'False'; ExternalVisible := 'False'; ExternalWritable := 'False'; S7_SetPoint := 'True'} : TP_TIME;   // Timer
      CheckActiveHMI_2 { ExternalAccessible := 'False'; ExternalVisible := 'False'; ExternalWritable := 'False'; S7_SetPoint := 'True'} : TON_TIME;   // Timer
      CheckActiveHMI_3 { ExternalAccessible := 'False'; ExternalVisible := 'False'; ExternalWritable := 'False'; S7_SetPoint := 'True'} : TON_TIME;   // Timer
   END_VAR
BEGIN

NETWORK
TITLE = **** 1 - Inputs **** DB number
// DB number
      L     DINO;
      T     #DBnr;

REGION Network 2: **** 1 - Inputs **** Extract the command bits from HMI
   // Extract the command bits from HMI
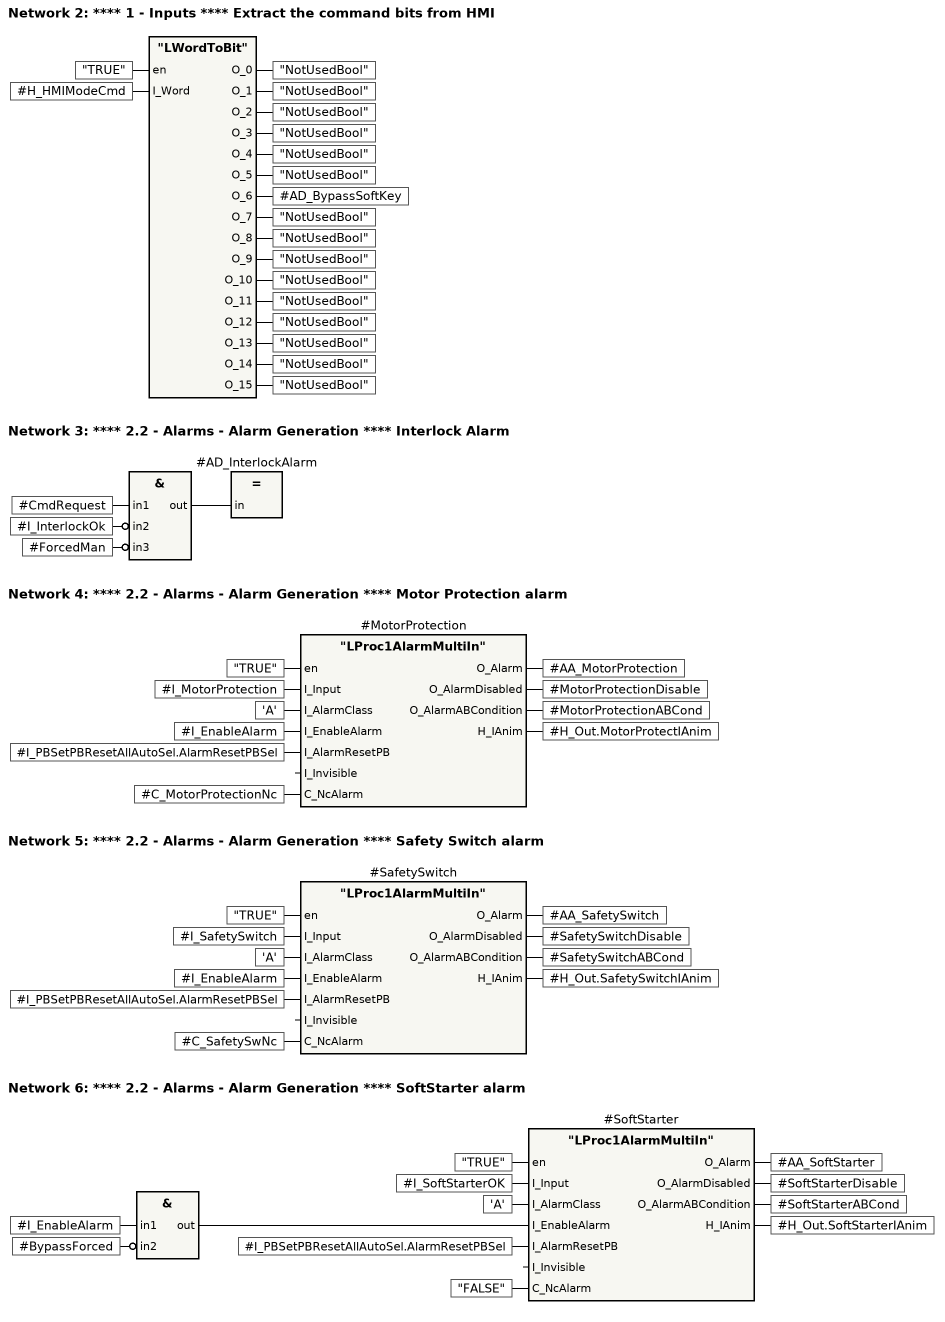
   IF "TRUE" THEN
       "LWordToBit"(I_Word := #H_HMIModeCmd,
                    O_0 => "NotUsedBool",
                    O_1 => "NotUsedBool",
                    O_2 => "NotUsedBool",
                    O_3 => "NotUsedBool",
                    O_4 => "NotUsedBool",
                    O_5 => "NotUsedBool",
                    O_6 => #AD_BypassSoftKey,
                    O_7 => "NotUsedBool",
                    O_8 => "NotUsedBool",
                    O_9 => "NotUsedBool",
                    O_10 => "NotUsedBool",
                    O_11 => "NotUsedBool",
                    O_12 => "NotUsedBool",
                    O_13 => "NotUsedBool",
                    O_14 => "NotUsedBool",
                    O_15 => "NotUsedBool");
   END_IF;
END_REGION

REGION Network 3: **** 2.2 - Alarms - Alarm Generation **** Interlock Alarm
   // Interlock Alarm
   #AD_InterlockAlarm := #CmdRequest AND NOT #I_InterlockOk AND NOT #ForcedMan;
END_REGION

REGION Network 4: **** 2.2 - Alarms - Alarm Generation **** Motor Protection alarm
   // Motor Protection alarm
   IF "TRUE" THEN
       #MotorProtection(I_Input := #I_MotorProtection,   // "LProc1AlarmMultiIn"
                        I_AlarmClass := 'A',
                        I_EnableAlarm := #I_EnableAlarm,
                        I_AlarmResetPB := #I_PBSetPBResetAllAutoSel.AlarmResetPBSel,
                        C_NcAlarm := #C_MotorProtectionNc,
                        O_Alarm => #AA_MotorProtection,
                        O_AlarmDisabled => #MotorProtectionDisable,
                        O_AlarmABCondition => #MotorProtectionABCond,
                        H_IAnim => #H_Out.MotorProtectIAnim);
   END_IF;
END_REGION

REGION Network 5: **** 2.2 - Alarms - Alarm Generation **** Safety Switch alarm
   // Safety Switch alarm
   IF "TRUE" THEN
       #SafetySwitch(I_Input := #I_SafetySwitch,   // "LProc1AlarmMultiIn"
                     I_AlarmClass := 'A',
                     I_EnableAlarm := #I_EnableAlarm,
                     I_AlarmResetPB := #I_PBSetPBResetAllAutoSel.AlarmResetPBSel,
                     C_NcAlarm := #C_SafetySwNc,
                     O_Alarm => #AA_SafetySwitch,
                     O_AlarmDisabled => #SafetySwitchDisable,
                     O_AlarmABCondition => #SafetySwitchABCond,
                     H_IAnim => #H_Out.SafetySwitchIAnim);
   END_IF;
END_REGION

REGION Network 6: **** 2.2 - Alarms - Alarm Generation **** SoftStarter alarm
   // SoftStarter alarm
   IF "TRUE" THEN
       #SoftStarter(I_Input := #I_SoftStarterOK,   // "LProc1AlarmMultiIn"
                    I_AlarmClass := 'A',
                    I_EnableAlarm := #I_EnableAlarm AND NOT #BypassForced,
                    I_AlarmResetPB := #I_PBSetPBResetAllAutoSel.AlarmResetPBSel,
                    C_NcAlarm := "FALSE",
                    O_Alarm => #AA_SoftStarter,
                    O_AlarmDisabled => #SoftStarterDisable,
                    O_AlarmABCondition => #SoftStarterABCond,
                    H_IAnim => #H_Out.SoftStarterIAnim);
   END_IF;
END_REGION

REGION Network 7: **** 2.2 - Alarms - Alarm Generation **** Bypass Switch alarm
   // Bypass Switch alarm
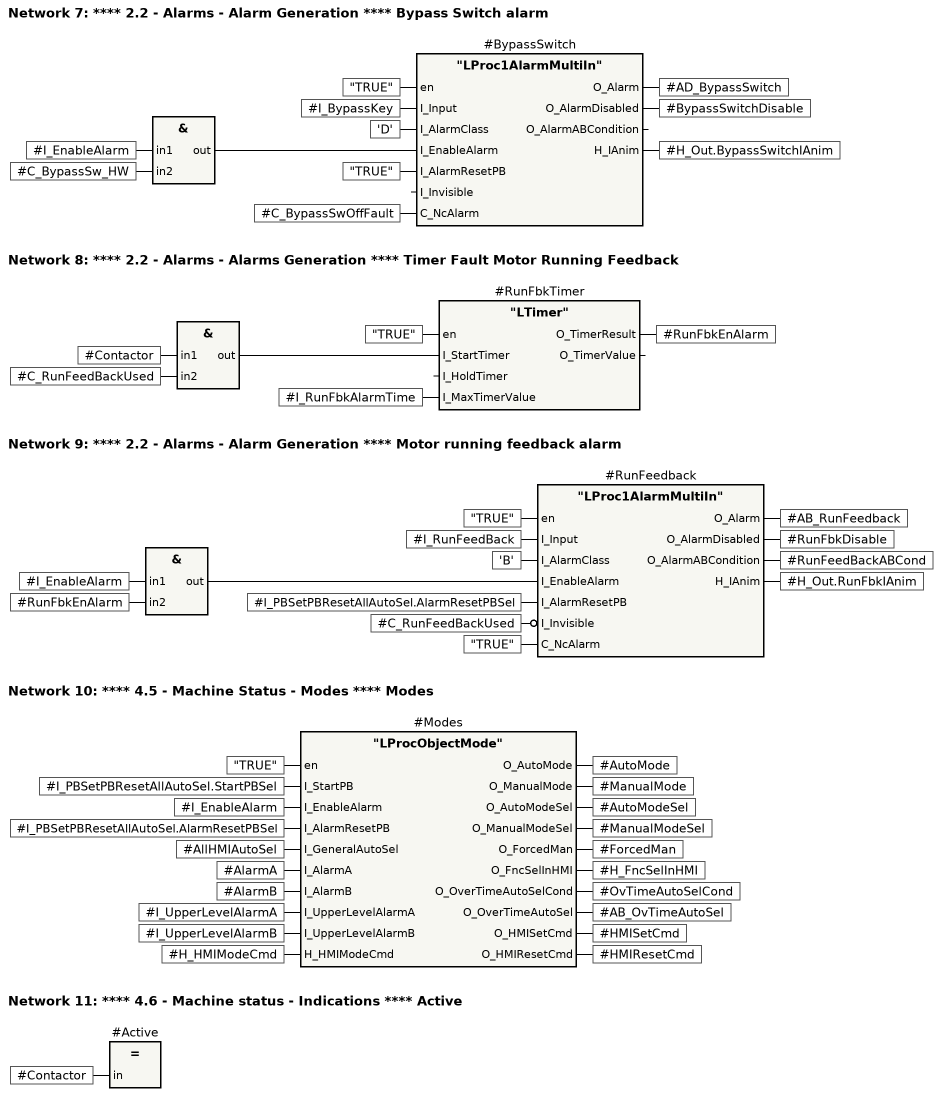
   IF "TRUE" THEN
       #BypassSwitch(I_Input := #I_BypassKey,   // "LProc1AlarmMultiIn"
                     I_AlarmClass := 'D',
                     I_EnableAlarm := #I_EnableAlarm AND #C_BypassSw_HW,
                     I_AlarmResetPB := "TRUE",
                     C_NcAlarm := #C_BypassSwOffFault,
                     O_Alarm => #AD_BypassSwitch,
                     O_AlarmDisabled => #BypassSwitchDisable,
                     H_IAnim => #H_Out.BypassSwitchIAnim);
   END_IF;
END_REGION

REGION Network 8: **** 2.2 - Alarms - Alarms Generation **** Timer Fault Motor Running Feedback
   // Timer Fault Motor Running Feedback
   IF "TRUE" THEN
       #RunFbkTimer(I_StartTimer := #Contactor AND #C_RunFeedBackUsed,   // "LTimer"
                    I_MaxTimerValue := #I_RunFbkAlarmTime,
                    O_TimerResult => #RunFbkEnAlarm);
   END_IF;
END_REGION

REGION Network 9: **** 2.2 - Alarms - Alarm Generation **** Motor running feedback alarm
   // Motor running feedback alarm
   IF "TRUE" THEN
       #RunFeedback(I_Input := #I_RunFeedBack,   // "LProc1AlarmMultiIn"
                    I_AlarmClass := 'B',
                    I_EnableAlarm := #I_EnableAlarm AND #RunFbkEnAlarm,
                    I_AlarmResetPB := #I_PBSetPBResetAllAutoSel.AlarmResetPBSel,
                    I_Invisible := NOT #C_RunFeedBackUsed,
                    C_NcAlarm := "TRUE",
                    O_Alarm => #AB_RunFeedback,
                    O_AlarmDisabled => #RunFbkDisable,
                    O_AlarmABCondition => #RunFeedBackABCond,
                    H_IAnim => #H_Out.RunFbkIAnim);
   END_IF;
END_REGION

REGION Network 10: **** 4.5 - Machine Status - Modes **** Modes
   // Modes
   IF "TRUE" THEN
       #Modes(I_StartPB := #I_PBSetPBResetAllAutoSel.StartPBSel,   // "LProcObjectMode"
              I_EnableAlarm := #I_EnableAlarm,
              I_AlarmResetPB := #I_PBSetPBResetAllAutoSel.AlarmResetPBSel,
              I_GeneralAutoSel := #AllHMIAutoSel,
              I_AlarmA := #AlarmA,
              I_AlarmB := #AlarmB,
              I_UpperLevelAlarmA := #I_UpperLevelAlarmA,
              I_UpperLevelAlarmB := #I_UpperLevelAlarmB,
              H_HMIModeCmd := #H_HMIModeCmd,
              O_AutoMode => #AutoMode,
              O_ManualMode => #ManualMode,
              O_AutoModeSel => #AutoModeSel,
              O_ManualModeSel => #ManualModeSel,
              O_ForcedMan => #ForcedMan,
              O_FncSelInHMI => #H_FncSelInHMI,
              O_OverTimeAutoSelCond => #OvTimeAutoSelCond,
              O_OverTimeAutoSel => #AB_OvTimeAutoSel,
              O_HMISetCmd => #HMISetCmd,
              O_HMIResetCmd => #HMIResetCmd);
   END_IF;
END_REGION

REGION Network 11: **** 4.6 - Machine status - Indications **** Active
   // Active
   #Active := #Contactor;
END_REGION

REGION Network 12: **** 4.6 - Machine status - Indications **** Contactor animation
   // Contactor animation
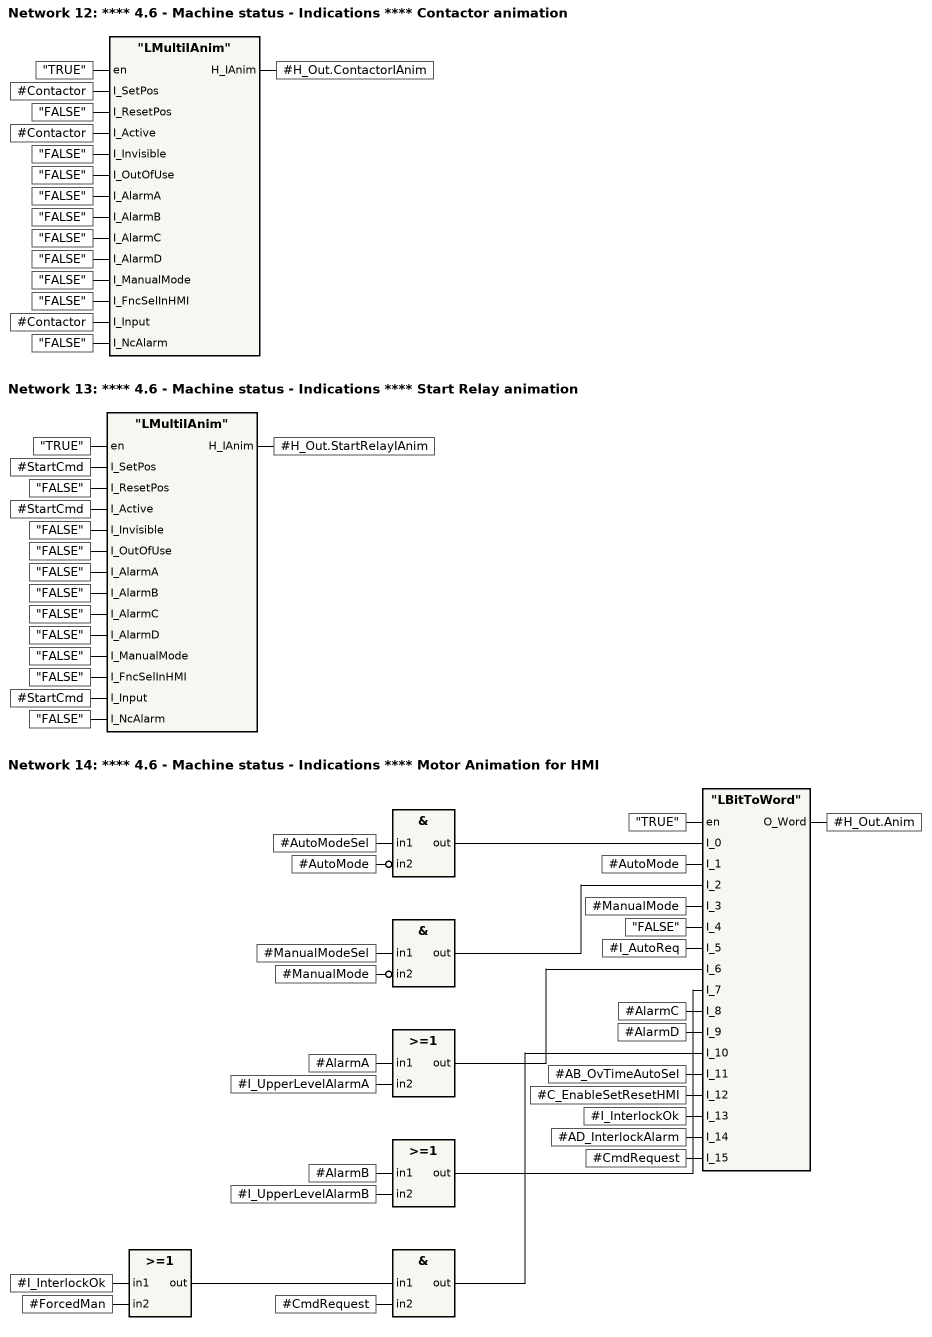
   IF "TRUE" THEN
       "LMultiIAnim"(I_SetPos := #Contactor,
                     I_ResetPos := "FALSE",
                     I_Active := #Contactor,
                     I_Invisible := "FALSE",
                     I_OutOfUse := "FALSE",
                     I_AlarmA := "FALSE",
                     I_AlarmB := "FALSE",
                     I_AlarmC := "FALSE",
                     I_AlarmD := "FALSE",
                     I_ManualMode := "FALSE",
                     I_FncSelInHMI := "FALSE",
                     I_Input := #Contactor,
                     I_NcAlarm := "FALSE",
                     H_IAnim => #H_Out.ContactorIAnim);
   END_IF;
END_REGION

REGION Network 13: **** 4.6 - Machine status - Indications **** Start Relay animation
   // Start Relay animation
   IF "TRUE" THEN
       "LMultiIAnim"(I_SetPos := #StartCmd,
                     I_ResetPos := "FALSE",
                     I_Active := #StartCmd,
                     I_Invisible := "FALSE",
                     I_OutOfUse := "FALSE",
                     I_AlarmA := "FALSE",
                     I_AlarmB := "FALSE",
                     I_AlarmC := "FALSE",
                     I_AlarmD := "FALSE",
                     I_ManualMode := "FALSE",
                     I_FncSelInHMI := "FALSE",
                     I_Input := #StartCmd,
                     I_NcAlarm := "FALSE",
                     H_IAnim => #H_Out.StartRelayIAnim);
   END_IF;
END_REGION

REGION Network 14: **** 4.6 - Machine status - Indications **** Motor Animation for HMI
   // Motor Animation for HMI
   IF "TRUE" THEN
       "LBitToWord"(I_0 := #AutoModeSel AND NOT #AutoMode,
                    I_1 := #AutoMode,
                    I_2 := #ManualModeSel AND NOT #ManualMode,
                    I_3 := #ManualMode,
                    I_4 := "FALSE",
                    I_5 := #I_AutoReq,
                    I_6 := #AlarmA OR #I_UpperLevelAlarmA,
                    I_7 := #AlarmB OR #I_UpperLevelAlarmB,
                    I_8 := #AlarmC,
                    I_9 := #AlarmD,
                    I_10 := (#I_InterlockOk OR #ForcedMan) AND #CmdRequest,
                    I_11 := #AB_OvTimeAutoSel,
                    I_12 := #C_EnableSetResetHMI,
                    I_13 := #I_InterlockOk,
                    I_14 := #AD_InterlockAlarm,
                    I_15 := #CmdRequest,
                    O_Word => #H_Out.Anim);
   END_IF;
END_REGION

REGION Network 15: **** 4.6 - Machine status - Indications **** Motor Animation for HMI
   // Motor Animation for HMI
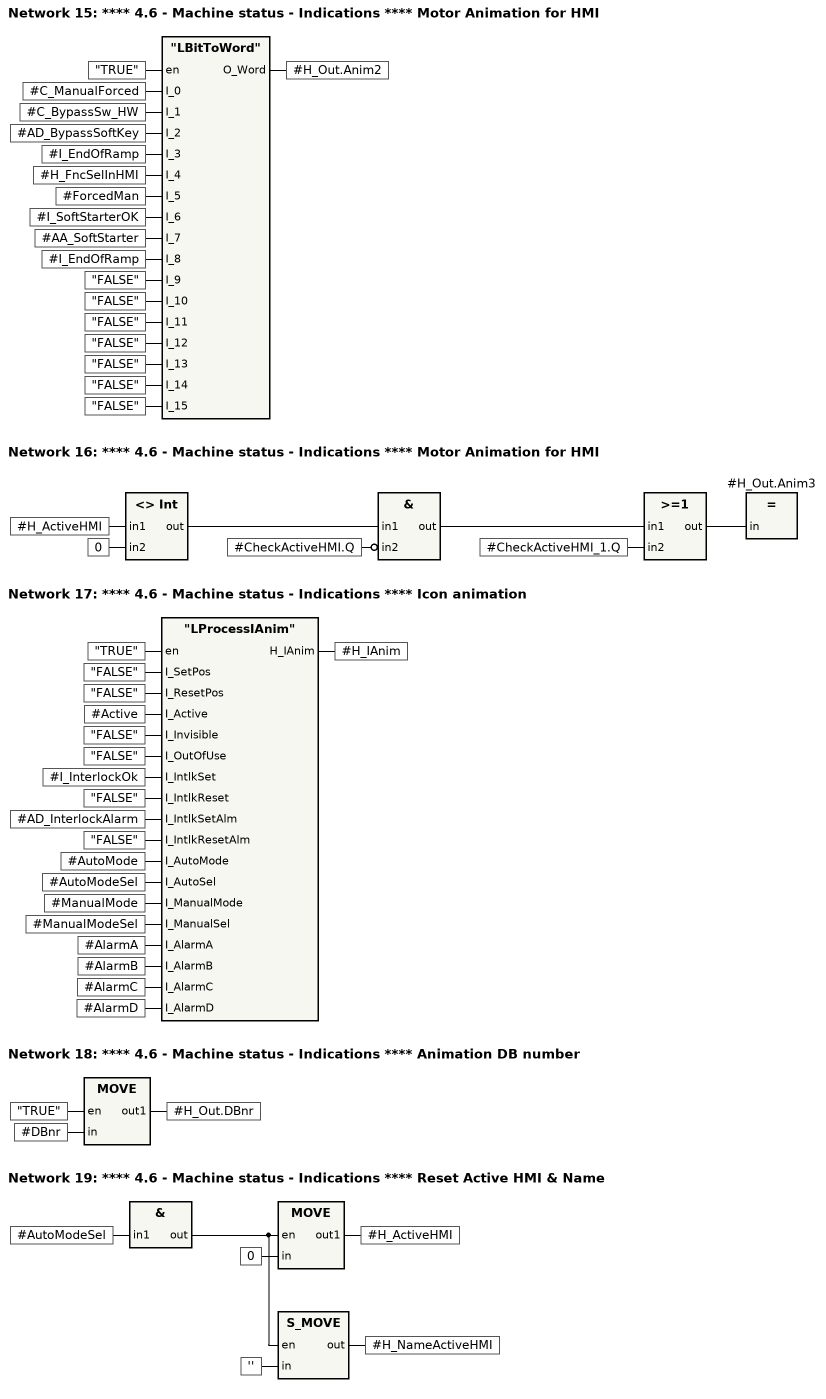
   IF "TRUE" THEN
       "LBitToWord"(I_0 := #C_ManualForced,
                    I_1 := #C_BypassSw_HW,
                    I_2 := #AD_BypassSoftKey,
                    I_3 := #I_EndOfRamp,
                    I_4 := #H_FncSelInHMI,
                    I_5 := #ForcedMan,
                    I_6 := #I_SoftStarterOK,
                    I_7 := #AA_SoftStarter,
                    I_8 := #I_EndOfRamp,
                    I_9 := "FALSE",
                    I_10 := "FALSE",
                    I_11 := "FALSE",
                    I_12 := "FALSE",
                    I_13 := "FALSE",
                    I_14 := "FALSE",
                    I_15 := "FALSE",
                    O_Word => #H_Out.Anim2);
   END_IF;
END_REGION

REGION Network 16: **** 4.6 - Machine status - Indications **** Motor Animation for HMI
   // Motor Animation for HMI
   #H_Out.Anim3 := ((#H_ActiveHMI <> 0) AND NOT #CheckActiveHMI.Q) OR #CheckActiveHMI_1.Q;
END_REGION

REGION Network 17: **** 4.6 - Machine status - Indications **** Icon animation
   // Icon animation
   IF "TRUE" THEN
       "LProcessIAnim"(I_SetPos := "FALSE",
                       I_ResetPos := "FALSE",
                       I_Active := #Active,
                       I_Invisible := "FALSE",
                       I_OutOfUse := "FALSE",
                       I_IntlkSet := #I_InterlockOk,
                       I_IntlkReset := "FALSE",
                       I_IntlkSetAlm := #AD_InterlockAlarm,
                       I_IntlkResetAlm := "FALSE",
                       I_AutoMode := #AutoMode,
                       I_AutoSel := #AutoModeSel,
                       I_ManualMode := #ManualMode,
                       I_ManualSel := #ManualModeSel,
                       I_AlarmA := #AlarmA,
                       I_AlarmB := #AlarmB,
                       I_AlarmC := #AlarmC,
                       I_AlarmD := #AlarmD,
                       H_IAnim => #H_IAnim);
   END_IF;
END_REGION

REGION Network 18: **** 4.6 - Machine status - Indications **** Animation DB number
   // Animation DB number
   IF "TRUE" THEN #H_Out.DBnr := #DBnr; END_IF;
END_REGION

REGION Network 19: **** 4.6 - Machine status - Indications **** Reset Active HMI & Name
   // Reset Active HMI & Name
   IF #AutoModeSel THEN
       #H_ActiveHMI := 0;
       #H_NameActiveHMI := '';
   END_IF;
END_REGION

REGION Network 20: **** 5.2 - Equations - Flow **** Manual mode is active and the Set button is pressed
   // Manual mode is active and the Set button is pressed
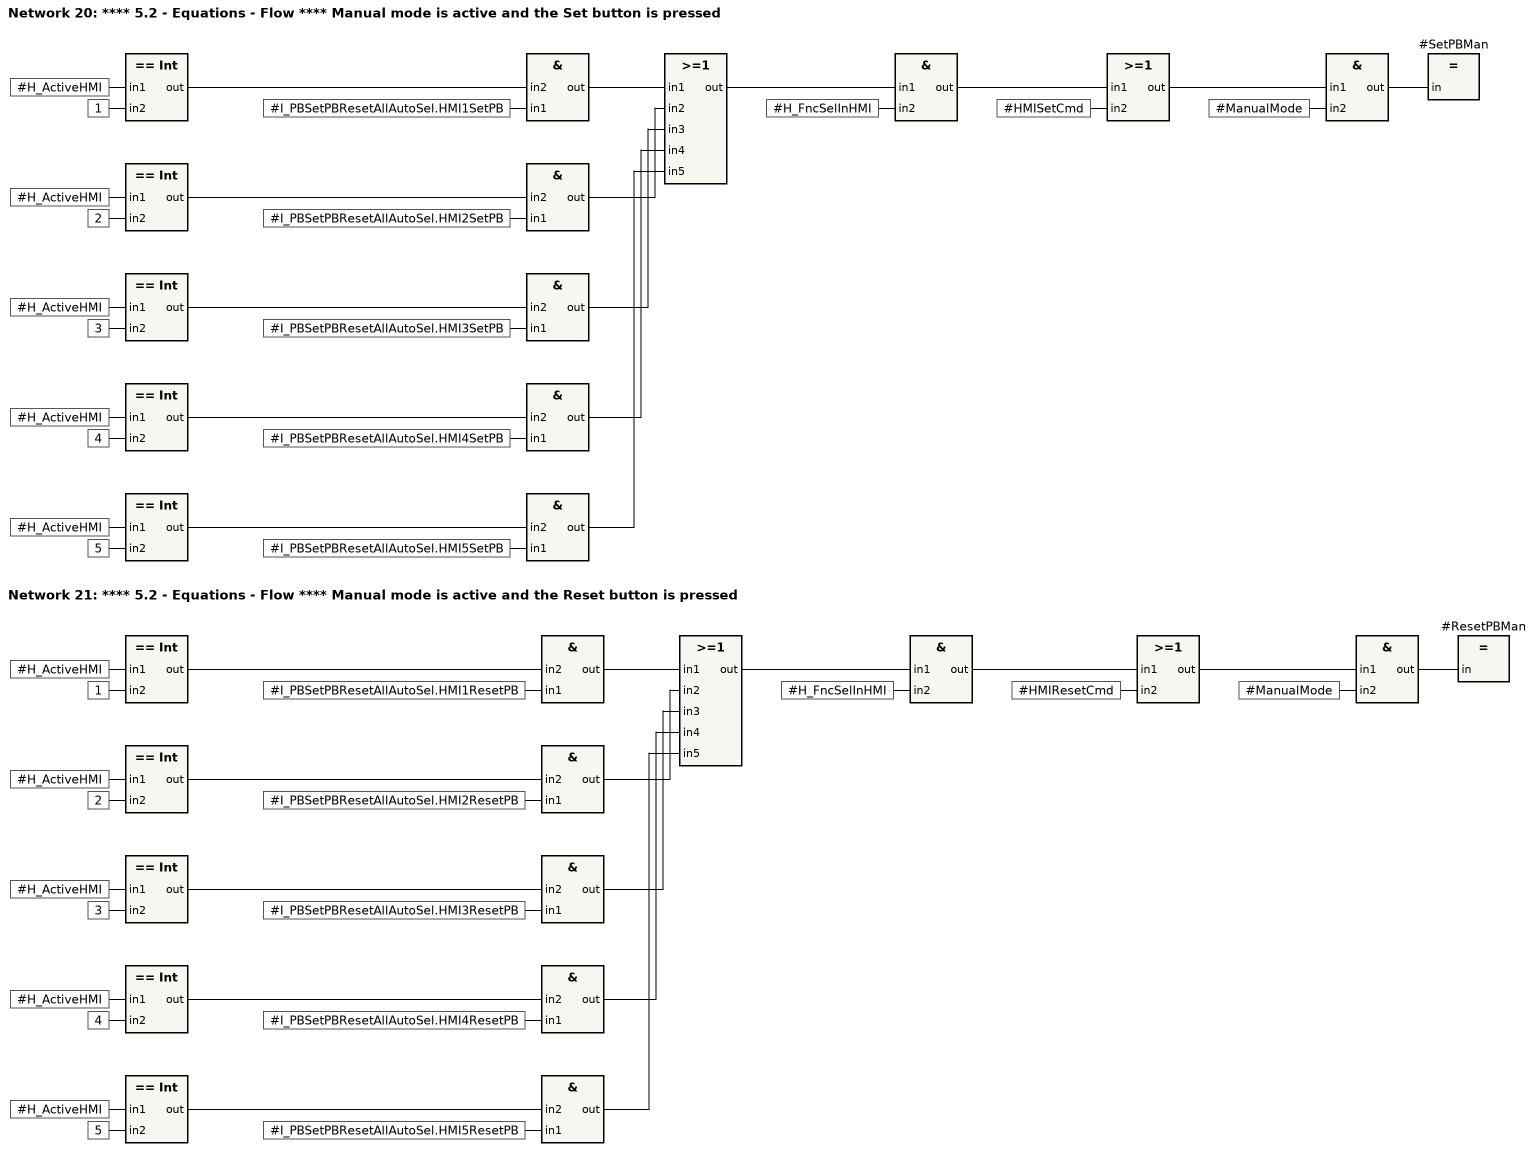
   #SetPBMan := (((((#H_ActiveHMI = 1) AND #I_PBSetPBResetAllAutoSel.HMI1SetPB) OR ((#H_ActiveHMI = 2) AND #I_PBSetPBResetAllAutoSel.HMI2SetPB) OR ((#H_ActiveHMI = 3) AND #I_PBSetPBResetAllAutoSel.HMI3SetPB) OR ((#H_ActiveHMI = 4) AND #I_PBSetPBResetAllAutoSel.HMI4SetPB) OR ((#H_ActiveHMI = 5) AND #I_PBSetPBResetAllAutoSel.HMI5SetPB)) AND #H_FncSelInHMI) OR #HMISetCmd) AND #ManualMode;
END_REGION

REGION Network 21: **** 5.2 - Equations - Flow **** Manual mode is active and the Reset button is pressed
   // Manual mode is active and the Reset button is pressed
   #ResetPBMan := (((((#H_ActiveHMI = 1) AND #I_PBSetPBResetAllAutoSel.HMI1ResetPB) OR ((#H_ActiveHMI = 2) AND #I_PBSetPBResetAllAutoSel.HMI2ResetPB) OR ((#H_ActiveHMI = 3) AND #I_PBSetPBResetAllAutoSel.HMI3ResetPB) OR ((#H_ActiveHMI = 4) AND #I_PBSetPBResetAllAutoSel.HMI4ResetPB) OR ((#H_ActiveHMI = 5) AND #I_PBSetPBResetAllAutoSel.HMI5ResetPB)) AND #H_FncSelInHMI) OR #HMIResetCmd) AND #ManualMode;
END_REGION

REGION Network 22: **** 5.2 - Equations - Flow **** All HMI Auto selected
   // All HMI Auto selected
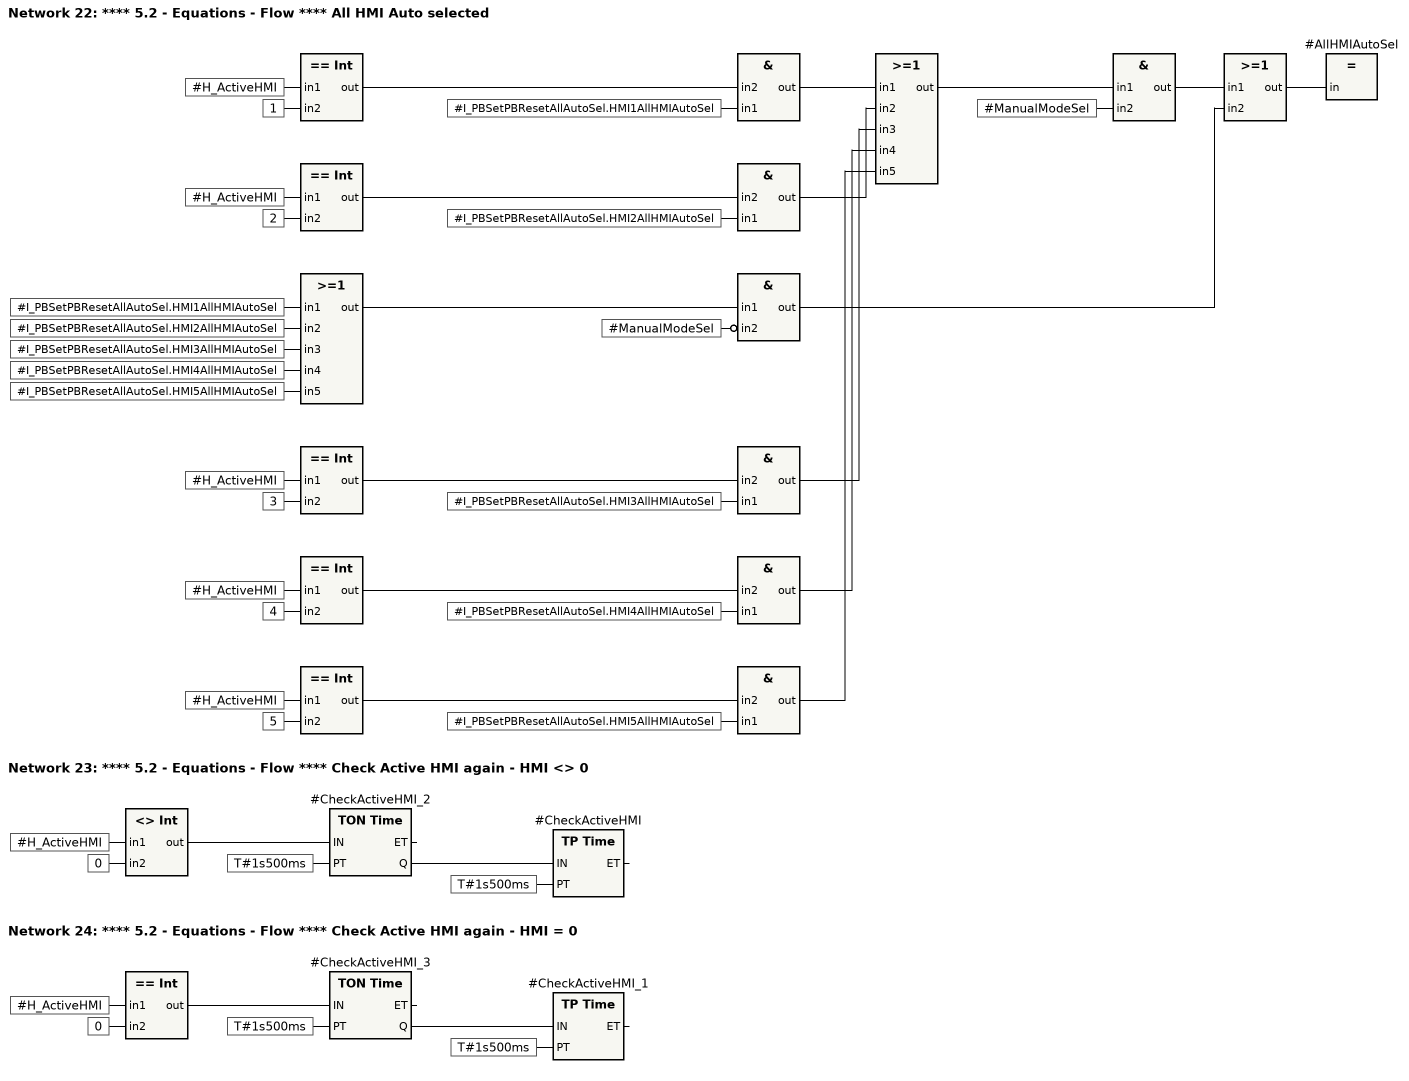
   #AllHMIAutoSel := ((((#H_ActiveHMI = 1) AND #I_PBSetPBResetAllAutoSel.HMI1AllHMIAutoSel) OR ((#H_ActiveHMI = 2) AND #I_PBSetPBResetAllAutoSel.HMI2AllHMIAutoSel) OR ((#H_ActiveHMI = 3) AND #I_PBSetPBResetAllAutoSel.HMI3AllHMIAutoSel) OR ((#H_ActiveHMI = 4) AND #I_PBSetPBResetAllAutoSel.HMI4AllHMIAutoSel) OR ((#H_ActiveHMI = 5) AND #I_PBSetPBResetAllAutoSel.HMI5AllHMIAutoSel)) AND #ManualModeSel) OR ((#I_PBSetPBResetAllAutoSel.HMI1AllHMIAutoSel OR #I_PBSetPBResetAllAutoSel.HMI2AllHMIAutoSel OR #I_PBSetPBResetAllAutoSel.HMI3AllHMIAutoSel OR #I_PBSetPBResetAllAutoSel.HMI4AllHMIAutoSel OR #I_PBSetPBResetAllAutoSel.HMI5AllHMIAutoSel) AND NOT #ManualModeSel);
END_REGION

REGION Network 23: **** 5.2 - Equations - Flow **** Check Active HMI again - HMI <> 0
   // Check Active HMI again
   #CheckActiveHMI_2(IN := #H_ActiveHMI <> 0, PT := T#1s500ms);   // TON
   #CheckActiveHMI(IN := #CheckActiveHMI_2.Q, PT := T#1s500ms);   // TP
END_REGION

REGION Network 24: **** 5.2 - Equations - Flow **** Check Active HMI again - HMI = 0
   // Check Active HMI again
   #CheckActiveHMI_3(IN := #H_ActiveHMI = 0, PT := T#1s500ms);   // TON
   #CheckActiveHMI_1(IN := #CheckActiveHMI_3.Q, PT := T#1s500ms);   // TP
END_REGION

REGION Network 25: **** 7.3 - Submodule - Machine **** Command Request
   // Command Request
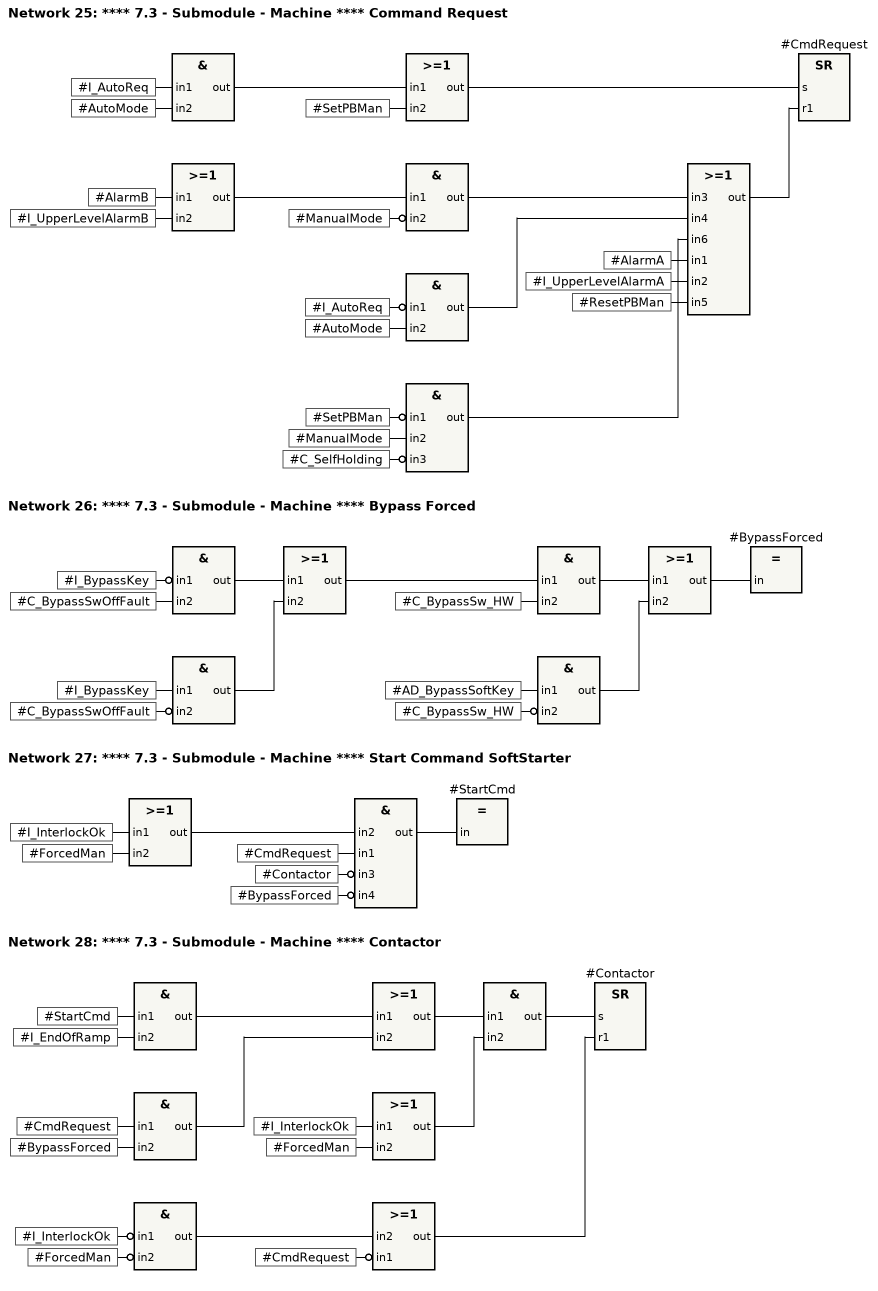
   IF (#I_AutoReq AND #AutoMode) OR #SetPBMan THEN
       #CmdRequest := TRUE;   // SR flip-flop
   END_IF;
   IF ((#AlarmB OR #I_UpperLevelAlarmB) AND NOT #ManualMode) OR (NOT #I_AutoReq AND #AutoMode) OR (NOT #SetPBMan AND #ManualMode AND NOT #C_SelfHolding) OR #AlarmA OR #I_UpperLevelAlarmA OR #ResetPBMan THEN
       #CmdRequest := FALSE;
   END_IF;
END_REGION

REGION Network 26: **** 7.3 - Submodule - Machine **** Bypass Forced
   // Bypass Forced
   #BypassForced := (((NOT #I_BypassKey AND #C_BypassSwOffFault) OR (#I_BypassKey AND NOT #C_BypassSwOffFault)) AND #C_BypassSw_HW) OR (#AD_BypassSoftKey AND NOT #C_BypassSw_HW);
END_REGION

REGION Network 27: **** 7.3 - Submodule - Machine **** Start Command SoftStarter
   // Start Command SoftStarter
   #StartCmd := (#I_InterlockOk OR #ForcedMan) AND #CmdRequest AND NOT #Contactor AND NOT #BypassForced;
END_REGION

REGION Network 28: **** 7.3 - Submodule - Machine **** Contactor
   // Contactor
   IF ((#StartCmd AND #I_EndOfRamp) OR (#CmdRequest AND #BypassForced)) AND (#I_InterlockOk OR #ForcedMan) THEN
       #Contactor := TRUE;   // SR flip-flop
   END_IF;
   IF (NOT #I_InterlockOk AND NOT #ForcedMan) OR NOT #CmdRequest THEN #Contactor := FALSE; END_IF;
END_REGION

REGION Network 29: **** 8 - Outputs **** Start Command SoftStarter
   // Start Command SoftStarter
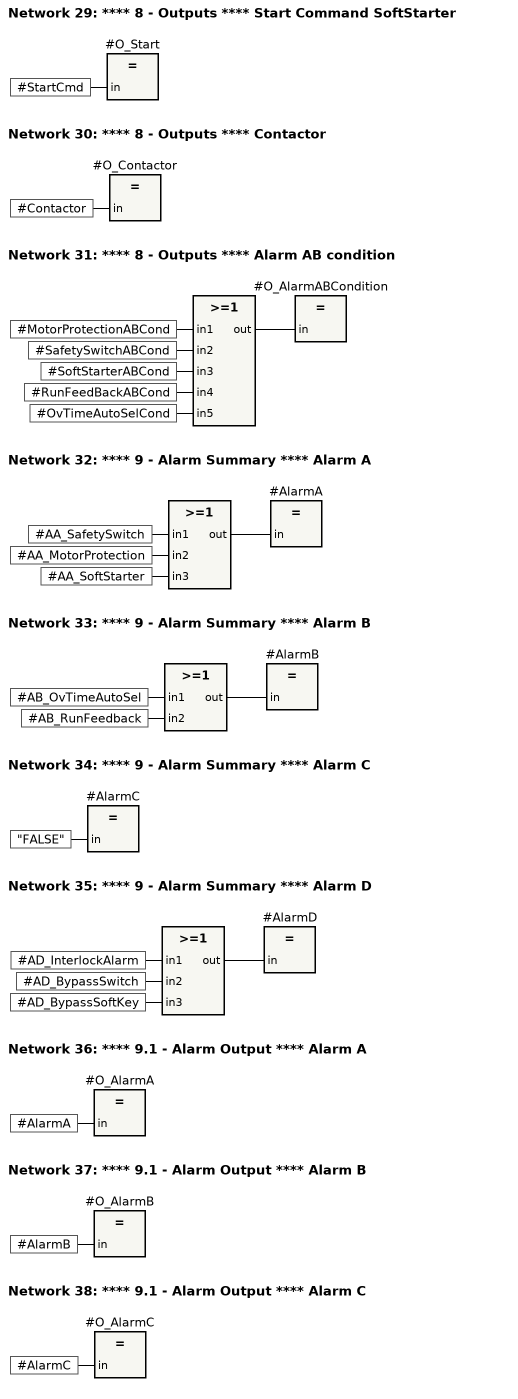
   #O_Start := #StartCmd;
END_REGION

REGION Network 30: **** 8 - Outputs **** Contactor
   // Contactor
   #O_Contactor := #Contactor;
END_REGION

REGION Network 31: **** 8 - Outputs **** Alarm AB condition
   // Alarm AB Condition
   #O_AlarmABCondition := #MotorProtectionABCond OR #SafetySwitchABCond OR #SoftStarterABCond OR #RunFeedBackABCond OR #OvTimeAutoSelCond;
END_REGION

REGION Network 32: **** 9 - Alarm Summary **** Alarm A
   // Alarm A
   #AlarmA := #AA_SafetySwitch OR #AA_MotorProtection OR #AA_SoftStarter;
END_REGION

REGION Network 33: **** 9 - Alarm Summary **** Alarm B
   // Alarm B
   #AlarmB := #AB_OvTimeAutoSel OR #AB_RunFeedback;
END_REGION

REGION Network 34: **** 9 - Alarm Summary **** Alarm C
   // Alarm C
   #AlarmC := "FALSE";
END_REGION

REGION Network 35: **** 9 - Alarm Summary **** Alarm D
   // Alarm D
   #AlarmD := #AD_InterlockAlarm OR #AD_BypassSwitch OR #AD_BypassSoftKey;
END_REGION

REGION Network 36: **** 9.1 - Alarm Output **** Alarm A
   // Alarm A
   #O_AlarmA := #AlarmA;
END_REGION

REGION Network 37: **** 9.1 - Alarm Output **** Alarm B
   // Alarm B
   #O_AlarmB := #AlarmB;
END_REGION

REGION Network 38: **** 9.1 - Alarm Output **** Alarm C
   // Alarm C
   #O_AlarmC := #AlarmC;
END_REGION

REGION Network 39: **** 9.1 - Alarm Output **** Alarm D
   // Alarm D
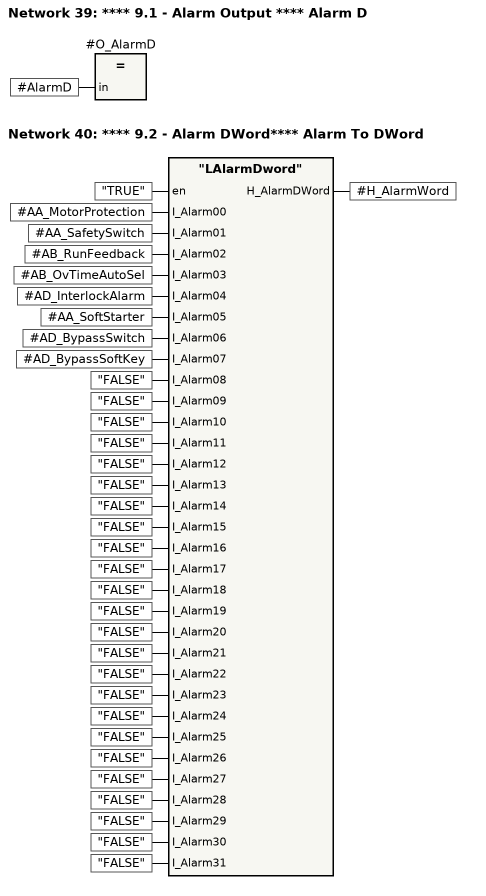
   #O_AlarmD := #AlarmD;
END_REGION

REGION Network 40: **** 9.2 - Alarm DWord**** Alarm To DWord
   // Alarm Word
   IF "TRUE" THEN
       "LAlarmDword"(I_Alarm00 := #AA_MotorProtection,
                     I_Alarm01 := #AA_SafetySwitch,
                     I_Alarm02 := #AB_RunFeedback,
                     I_Alarm03 := #AB_OvTimeAutoSel,
                     I_Alarm04 := #AD_InterlockAlarm,
                     I_Alarm05 := #AA_SoftStarter,
                     I_Alarm06 := #AD_BypassSwitch,
                     I_Alarm07 := #AD_BypassSoftKey,
                     I_Alarm08 := "FALSE",
                     I_Alarm09 := "FALSE",
                     I_Alarm10 := "FALSE",
                     I_Alarm11 := "FALSE",
                     I_Alarm12 := "FALSE",
                     I_Alarm13 := "FALSE",
                     I_Alarm14 := "FALSE",
                     I_Alarm15 := "FALSE",
                     I_Alarm16 := "FALSE",
                     I_Alarm17 := "FALSE",
                     I_Alarm18 := "FALSE",
                     I_Alarm19 := "FALSE",
                     I_Alarm20 := "FALSE",
                     I_Alarm21 := "FALSE",
                     I_Alarm22 := "FALSE",
                     I_Alarm23 := "FALSE",
                     I_Alarm24 := "FALSE",
                     I_Alarm25 := "FALSE",
                     I_Alarm26 := "FALSE",
                     I_Alarm27 := "FALSE",
                     I_Alarm28 := "FALSE",
                     I_Alarm29 := "FALSE",
                     I_Alarm30 := "FALSE",
                     I_Alarm31 := "FALSE",
                     H_AlarmDWord => #H_AlarmWord);
   END_IF;
END_REGION
END_FUNCTION_BLOCK

FUNCTION_BLOCK "LProcDO_Fbk"   // FB1717, FBD
TITLE = LProcDO_Fbk
{ S7_Optimized_Access := 'FALSE' }
AUTHOR : VCC
FAMILY : ProcEq
NAME : DOFbk
VERSION : 0.1
// ================================================================================
// This module converts the signal 0-100% to digital commands Open and Close to 
// steer in position a valve or damper equipped with a motor.
// The controller is operating with the feedback for the position of the valve.
// Detections Open/Close may be connected to the controller to check the correct 
// opening and closing of the valve or damper.
// ================================================================================
// stored: AutoNumber false, IsIECCheckEnabled false, SetENOAutomatically False, UDAEnableTagReadback false
   VAR_INPUT
      I_CYCLE { ExternalAccessible := 'False'; ExternalVisible := 'False'; ExternalWritable := 'False'} : Time;   // Sample time
      H_PULSE_TM : Time;   // Minimum Pulse Time
      H_BREAK_TM : Time;   // Minimum Break Time
      I_SP : Real;   // Set-point Input
      H_DEADB_W : Real;   // Slave: Deadband width
      H_FAC : Real := 1.0;   // Factor for feedback position
      I_POS { ExternalAccessible := 'False'; ExternalVisible := 'False'; ExternalWritable := 'False'} : Int;   // Feedback Position Input
      I_COM_RST { ExternalAccessible := 'False'; ExternalVisible := 'False'; ExternalWritable := 'False'} : Bool;   // Initialising reset of controller
   END_VAR
   VAR_OUTPUT
      O_PosFbk { ExternalAccessible := 'False'; ExternalVisible := 'False'; ExternalWritable := 'False'} : Real;   // Output Feedback Position
      O_Set { ExternalAccessible := 'False'; ExternalVisible := 'False'; ExternalWritable := 'False'} : Bool;   // DO output Set
      O_Reset { ExternalAccessible := 'False'; ExternalVisible := 'False'; ExternalWritable := 'False'} : Bool;   // DO output Reset
   END_VAR
   VAR DB_SPECIFIC
      Pos { ExternalAccessible := 'False'; ExternalVisible := 'False'; ExternalWritable := 'False'} : Word;   // Feedback Position in WORD
   END_VAR
   VAR
      DO_Controller { ExternalAccessible := 'False'; ExternalVisible := 'False'; ExternalWritable := 'False'; S7_SetPoint := 'True'} : CONT_S;
   END_VAR
BEGIN

REGION Network 1: **** 5.2 - Equations - Flow Equations **** Convert Position from integer to word
   // Convert Position from integer to word
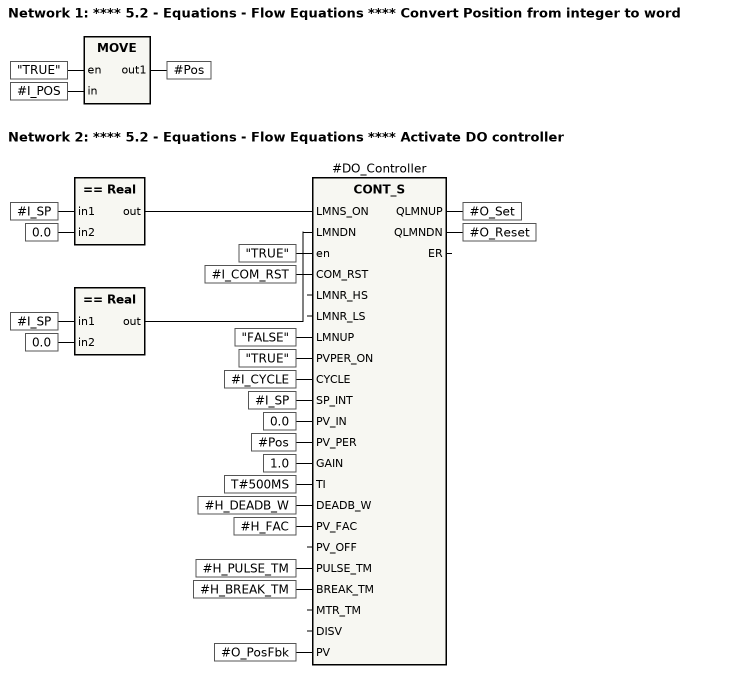
   IF "TRUE" THEN #Pos := #I_POS; END_IF;
END_REGION

REGION Network 2: **** 5.2 - Equations - Flow Equations **** Activate DO controller
   // Activate DO controller
   IF "TRUE" THEN
       #DO_Controller(LMNS_ON := #I_SP = 0.0,   // CONT_S
                      LMNDN := #I_SP = 0.0,
                      COM_RST := #I_COM_RST,
                      LMNUP := "FALSE",
                      PVPER_ON := "TRUE",
                      CYCLE := #I_CYCLE,
                      SP_INT := #I_SP,
                      PV_IN := 0.0,
                      PV_PER := #Pos,
                      GAIN := 1.0,
                      TI := T#500MS,
                      DEADB_W := #H_DEADB_W,
                      PV_FAC := #H_FAC,
                      PULSE_TM := #H_PULSE_TM,
                      BREAK_TM := #H_BREAK_TM,
                      PV := #O_PosFbk,
                      QLMNUP => #O_Set,
                      QLMNDN => #O_Reset);
   END_IF;
END_REGION
END_FUNCTION_BLOCK

FUNCTION_BLOCK "LProcEntalphie"   // FB1718, STL
TITLE = LProcEnthalpie
{ S7_Optimized_Access := 'FALSE' }
AUTHOR : VCC
FAMILY : ProcEq
VERSION : 0.1
// This function is made for the calculatin of the Ethalpie from the temperature 
// and humidity measurements.
// stored: AutoNumber false, UDAEnableTagReadback false
   VAR_INPUT
      PvHumidity { ExternalAccessible := 'False'; ExternalVisible := 'False'; ExternalWritable := 'False'} : Real;   // Analoge input value humidity
      PvTemperature { ExternalAccessible := 'False'; ExternalVisible := 'False'; ExternalWritable := 'False'} : Real;   // Analoge intup value temperature
   END_VAR
   VAR_OUTPUT
      PvEnthalpie { ExternalAccessible := 'False'; ExternalVisible := 'False'; ExternalWritable := 'False'} : Real;   // Enthalpy calculation
   END_VAR
   VAR DB_SPECIFIC
      PvX { ExternalAccessible := 'False'; ExternalVisible := 'False'; ExternalWritable := 'False'} : Real;   // Humidity absolute for the process value
      PvPs { ExternalAccessible := 'False'; ExternalVisible := 'False'; ExternalWritable := 'False'} : Real;   // Value for steam pressure for the humidity value
      PvNbXYpoints { ExternalAccessible := 'False'; ExternalVisible := 'False'; ExternalWritable := 'False'} : Int;   // Edit number of X-Y points used
      PvFraction { ExternalAccessible := 'False'; ExternalVisible := 'False'; ExternalWritable := 'False'} : Int;
      PvBias { ExternalAccessible := 'False'; ExternalVisible := 'False'; ExternalWritable := 'False'} : Real;
      xl { ExternalAccessible := 'False'; ExternalVisible := 'False'; ExternalWritable := 'False'} : Real;
      xh { ExternalAccessible := 'False'; ExternalVisible := 'False'; ExternalWritable := 'False'} : Real;
      yl { ExternalAccessible := 'False'; ExternalVisible := 'False'; ExternalWritable := 'False'} : Real;
      yh { ExternalAccessible := 'False'; ExternalVisible := 'False'; ExternalWritable := 'False'} : Real;
      PvPstemp1 { ExternalAccessible := 'False'; ExternalVisible := 'False'; ExternalWritable := 'False'} : Real;
      PvPsTemp2 { ExternalAccessible := 'False'; ExternalVisible := 'False'; ExternalWritable := 'False'} : Real;
      PvPsTemp3 { ExternalAccessible := 'False'; ExternalVisible := 'False'; ExternalWritable := 'False'} : Real;
      PvXTemp1 { ExternalAccessible := 'False'; ExternalVisible := 'False'; ExternalWritable := 'False'} : Real;
      PvxTemp2 { ExternalAccessible := 'False'; ExternalVisible := 'False'; ExternalWritable := 'False'} : Real;
      PvXTemp3 { ExternalAccessible := 'False'; ExternalVisible := 'False'; ExternalWritable := 'False'} : Real;
      PvEnthTemp1 { ExternalAccessible := 'False'; ExternalVisible := 'False'; ExternalWritable := 'False'} : Real;
      PvEnthTemp2 { ExternalAccessible := 'False'; ExternalVisible := 'False'; ExternalWritable := 'False'} : Real;
   END_VAR
BEGIN

NETWORK
TITLE = **** 4.4 - Machine status - Calculation **** Calculate position
// Calculate position
      L     -10.0;
      T     #xl;
      L     260.0;
      T     #yl;
      L     0.0;
      T     #xh;
      L     610.59;
      T     #yh;






NETWORK
TITLE = **** 4.4 - Machine status - Calculation **** Calculate position
// Calculate position
      A(;
      L     #PvTemperature;
      L     0.0;
      >R;
      );
      JCN   End1;
      L     #xh;
      T     #xl;
      L     #yh;
      T     #yl;
      L     6.0;
      T     #xh;
      L     934.59;
      T     #yh;

End1: NOP   0;





NETWORK
TITLE = **** 4.4 - Machine status - Calculation **** Calculate position
// Calculate position
      A(;
      L     #PvTemperature;
      L     6.0;
      >R;
      );
      JCN   End2;
      L     #xh;
      T     #xl;
      L     #yh;
      T     #yl;
      L     12.0;
      T     #xh;
      L     1402.5;
      T     #yh;

End2: NOP   0;




NETWORK
TITLE = **** 4.4 - Machine status - Calculation **** Calculate position
// Calculate position
      A(;
      L     #PvTemperature;
      L     12.0;
      >R;
      );
      JCN   End3;
      L     #xh;
      T     #xl;
      L     #yh;
      T     #yl;
      L     16.0;
      T     #xh;
      L     1817.2;
      T     #yh;

End3: NOP   0;





NETWORK
TITLE = **** 4.4 - Machine status - Calculation **** Calculate position
// Calculate position
      A(;
      L     #PvTemperature;
      L     16.0;
      >R;
      );
      JCN   End4;
      L     #xh;
      T     #xl;
      L     #yh;
      T     #yl;
      L     20.0;
      T     #xh;
      L     2337.1;
      T     #yh;

End4: NOP   0;





NETWORK
TITLE = **** 4.4 - Machine status - Calculation **** Calculate position
// Calculate position
      A(;
      L     #PvTemperature;
      L     20.0;
      >R;
      );
      JCN   End5;
      L     #xh;
      T     #xl;
      L     #yh;
      T     #yl;
      L     22.0;
      T     #xh;
      L     2643.8;
      T     #yh;

End5: NOP   0;




NETWORK
TITLE = **** 4.4 - Machine status - Calculation **** Calculate position
// Calculate position
      A(;
      L     #PvTemperature;
      L     22.0;
      >R;
      );
      JCN   End6;
      L     #xh;
      T     #xl;
      L     #yh;
      T     #yl;
      L     26.0;
      T     #xh;
      L     3361.0;
      T     #yh;

End6: NOP   0;





NETWORK
TITLE = **** 4.4 - Machine status - Calculation **** Calculate position
// Calculate position
      A(;
      L     #PvTemperature;
      L     26.0;
      >R;
      );
      JCN   End7;
      L     #xh;
      T     #xl;
      L     #yh;
      T     #yl;
      L     32.0;
      T     #xh;
      L     4754.3;
      T     #yh;

End7: NOP   0;





NETWORK
TITLE = **** 4.4 - Machine status - Calculation **** Calculate position
// Calculate position
      A(;
      L     #PvTemperature;
      L     32.0;
      >R;
      );
      JCN   End8;
      L     #xh;
      T     #xl;
      L     #yh;
      T     #yl;
      L     40.0;
      T     #xh;
      L     7375.4;
      T     #yh;

End8: NOP   0;




NETWORK
TITLE = **** 4.4 - Machine status - Calculation **** Process value Enthalpie
// Process value Enthalpie
      L     #xh;
      L     #xl;
      -R;
      ABS;
      L     0.0001;
      <R;
      JC    then;
      L     #yh;
      L     #yl;
      -R;
      T     #PvPstemp1;
      L     #xh;
      L     #xl;
      -R;
      T     #PvPsTemp2;
      L     #PvTemperature;
      L     #xl;
      -R;
      T     #PvPsTemp3;
      L     #PvPstemp1;
      L     #PvPsTemp2;
      /R;
      L     #PvPsTemp3;
      *R;
      L     #yl;
      +R;
      L     #PvBias;
      +R;
      T     #PvPs;
      JU    End;

then: L     #yh;
      L     #yl;
      +R;
      L     2.0;
      /R;
      L     #PvBias;
      +R;
      T     #PvPs;


End:  NOP   0;




NETWORK
TITLE = **** 4.4 - Machine status - Calculation **** Humidity absolut
// Humidity absolut
      L     0.622;
      L     #PvHumidity;
      *R;
      L     100.0;
      /R;
      L     #PvPs;
      *R;
      T     #PvXTemp1;
      L     #PvHumidity;
      L     100.0;
      /R;
      L     #PvPs;
      *R;
      T     #PvxTemp2;
      L     101356.9;
      L     #PvxTemp2;
      -R;
      T     #PvXTemp3;
      L     #PvXTemp1;
      L     #PvXTemp3;
      /R;
      T     #PvX;




NETWORK
TITLE = **** 4.4 - Machine status - Calculation **** Calculation of the process enthalpie value
// Calculation of the process enthalpie value
      L     2500.8;
      L     #PvX;
      *R;
      T     #PvEnthTemp1;
      L     1.927;
      L     #PvX;
      *R;
      L     #PvTemperature;
      *R;
      T     #PvEnthTemp2;
      L     1.006;
      L     #PvTemperature;
      *R;
      L     #PvEnthTemp1;
      +R;
      L     #PvEnthTemp2;
      +R;
      T     #PvEnthalpie;




END_FUNCTION_BLOCK

